bError:=fbReadVelocityToCam.bError OR fbReadVelocityFromCam.bError;
IF fbReadVelocityToCam.bError THEN
  nErrorId:=fbReadVelocityToCam.nErrorId;
ELSIF fbReadVelocityFromCam.bError THEN
  nErrorId:=fbReadVelocityFromCam.nErrorId;
END_IF

END_FUNCTION_BLOCK

// tc_mca_std_lib/POUs/ChangeConfig/FB_ReadFloatParameter
FUNCTION_BLOCK FB_ReadFloatParameter
VAR_INPUT
	bExecute: BOOL;
	///16#4000=Axisdata, 16#5000=Encoderdata, 16#6000=Controldata, 16#7000=Drivedata
	nDeviceGroup: UDINT;
	nIndexOffset: UDINT;
END_VAR
VAR_OUTPUT
	nData: LREAL;
	bBusy: BOOL;
	bDone: BOOL;
	bError: BOOL;
	nErrorId: UDINT;
END_VAR
VAR_IN_OUT
	Axis: AXIS_REF;
END_VAR
VAR
	nState: UINT;
	fbADSREAD: ADSREAD;
END_VAR

(*Sequence to read parameter in Nc*)
CASE nState OF
0:  (*Start sequence. Wait until bExecute is TRUE*)
	IF bExecute THEN
		bBusy:=TRUE;
		bError:=FALSE;
		nErrorId:=0;
		nState:=10;
	END_IF

10: (*Read parameter in Nc*)
	fbADSREAD(
		PORT:=500,
		IDXGRP:=nDeviceGroup+Axis.NcToPlc.AxisId,
		IDXOFFS:=nIndexOffset,
		LEN:=SIZEOF(nData),
		DESTADDR:=ADR(nData),
		READ:=TRUE);

	(*Wait until it's done or if an error occurs*)
	IF NOT fbADSREAD.ERR THEN
		IF NOT fbADSREAD.BUSY THEN
			fbADSREAD(READ:=FALSE);
			nState:=20;
		END_IF
	ELSE
		nErrorId:=fbADSREAD.ERRID;
		nState:=999;
	END_IF

20: (*Sequense is done. Waits until bExecute is FALSE*)
	bBusy:=FALSE;
	bDone:=TRUE;
	IF NOT bExecute THEN
		bDone:=FALSE;
		nState:=0;
	END_IF

999: (*Error in sequence*)
	bError:=TRUE;
	bBusy:=FALSE;
	bDone:=FALSE;
	fbADSREAD(READ:=FALSE);
	IF NOT bExecute THEN
		nState:=0;
	END_IF

END_CASE

END_FUNCTION_BLOCK

// tc_mca_std_lib/POUs/Motion/Homing/FB_HomeFinish
FUNCTION_BLOCK FB_HomeFinish
VAR_INPUT
	En: BOOL;
	bReset: BOOL;
    bExecute: BOOL;	
    nCmdData: UINT;
	bSofLimEnableLow: BOOL:=TRUE;
	bSofLimEnableHigh: BOOL:=TRUE;			
END_VAR
VAR_IN_OUT
	Axis: AXIS_REF;
END_VAR
VAR_OUTPUT
	EnO: BOOL;	
	bBusy: BOOL;
	bDone: BOOL;
	bError: BOOL;
	nErrorId: UDINT;
END_VAR
VAR		
	fbHomewriteSoftLimEnable:FB_HomeWriteSoftLimEnable;	
	fbExecuteRiseEdge: R_TRIG;	
	bExecuteWriteNC:BOOL:=FALSE;
	nState:INT:=0;
END_VAR

En:=EnO;
IF bReset THEN
	bError:=FALSE;
	nErrorId:=0;
END_IF 

IF NOT bExecute THEN
  bExecuteWriteNC:=FALSE;
  fbHomewriteSoftLimEnable.bSofLimEnableLow:=bSofLimEnableLow;
  fbHomewriteSoftLimEnable.bSofLimEnableHigh:=bSofLimEnableHigh;   
  nState:=0;
END_IF

fbExecuteRiseEdge(CLK:=bExecute);
IF fbExecuteRiseEdge.Q THEN
  bExecuteWriteNC:=TRUE;  
  fbHomewriteSoftLimEnable.bSofLimEnableLow:=bSofLimEnableLow;
  fbHomewriteSoftLimEnable.bSofLimEnableHigh:=bSofLimEnableHigh;
END_IF

// Write to NC (disable soft limits)
fbHomewriteSoftLimEnable(
	En:=En,
	bExecute:=bExecuteWriteNC AND bExecute,
	Axis:=Axis,
	bReset:=bReset,	
);

bBusy:=fbHomewriteSoftLimEnable.bBusy;
bDone:=fbHomewriteSoftLimEnable.bDone;

bError:=fbHomewriteSoftLimEnable.bError;
IF fbHomewriteSoftLimEnable.bError THEN
  nErrorId:=fbHomewriteSoftLimEnable.nErrorId;
END_IF

END_FUNCTION_BLOCK

// POUs/Motion/FB_MotionHoming
FUNCTION_BLOCK FB_MotionHoming
VAR_IN_OUT
    stMotionStage: DUT_MotionStage;
END_VAR
VAR_INPUT
    bExecute: BOOL;
END_VAR
VAR_OUTPUT
    bBusy: BOOL;
    bDone: BOOL;
    bError: BOOL;
    nErrorID: UDINT;
END_VAR
VAR
    fbSetPos: MC_SetPosition;
    fbJog: MC_Jog;
    rtExec: R_TRIG;
    ftExec: F_TRIG;
    nHomeStateMachine: INT := IDLE;
    nStateAfterStop: INT;
    nMoves: INT;
    bFirstDirection: BOOL;
    bAtHome: BOOL;
    bMove: BOOL;
    nErrCount: INT;
    bInterrupted: BOOL;
END_VAR
VAR CONSTANT
    IDLE: INT := 0;
    NEXT_MOVE: INT := 1;
    CHECK_FWD: INT := 2;
    CHECK_BWD: INT := 3;
    FINAL_MOVE: INT := 4;
    FINAL_SETPOS: INT := 5;
    ERROR: INT := 6;
    WAIT_STOP: INT := 7;

    (*
        This is a simpler way of disabling the soft limits that ends up being really obvious if something has gone wrong.
        If you turn the limits off/on, not only do you need to keep track of if you had soft limits set,
        but you need to always restore this properly or risk some issue.
        Instead, I set position to a ridiculous value that can always move forward or backward.
        If this gets stuck for any reason it's very clear that something has gone wrong,
        rather than a silent failure of the soft limit marks.
    *)
    FWD_START: LREAL := -99999999;
    BWD_START: LREAL :=  99999999;
END_VAR


fbSetPos.Options.ClearPositionLag := TRUE;
rtExec(CLK:=bExecute);
ftExec(CLK:=bExecute);

bError R= NOT bExecute;
IF NOT bError THEN
    nErrorID := 0;
END_IF

CASE stMotionStage.nHomingMode OF
    ENUM_EpicsHomeCmd.LOW_LIMIT:
        bFirstDirection := FALSE;
        bAtHome := NOT stMotionStage.bLimitBackwardEnable;
        bMove := TRUE;
    ENUM_EpicsHomeCmd.HIGH_LIMIT:
        bFirstDirection := TRUE;
        bAtHome := NOT stMotionStage.bLimitForwardEnable;
        bMove := TRUE;
    ENUM_EpicsHomeCmd.HOME_VIA_LOW:
        bFirstDirection := FALSE;
        bAtHome := stMotionStage.bHome;
        bMove := TRUE;
    ENUM_EpicsHomeCmd.HOME_VIA_HIGH:
        bFirstDirection := TRUE;
        bAtHome := stMotionStage.bHome;
        bMove := TRUE;
    ENUM_EpicsHomeCmd.ABSOLUTE_SET:
        fbSetPos(
            Axis:=stMotionStage.Axis,
            Execute:=bExecute,
            Position:=stMotionStage.fHomePosition);
        bBusy := rtExec.Q;
        bDone := NOT rtExec.Q;
        bMove := FALSE;
    ENUM_EpicsHomeCmd.NONE:
        bMove := FALSE;
        bBusy := rtExec.Q;
        bDone := NOT rtExec.Q;
    ELSE
        bMove := FALSE;
END_CASE

IF bMove THEN
    IF bBusy AND ftExec.Q THEN
        nHomeStateMachine := ERROR;
        bInterrupted := TRUE;
    END_IF
    CASE nHomeStateMachine OF
        // Wait for a rising edge
        IDLE:
            bBusy := FALSE;
            nErrCount := 0;
            fbSetPos(
                Axis:=stMotionStage.Axis,
                Execute:=FALSE);
            fbJog(
                Axis:=stMotionStage.Axis,
                JogForward:=FALSE,
                JogBackwards:=FALSE);
            IF rtExec.Q THEN
                nHomeStateMachine := NEXT_MOVE;
                nMoves := 0;
                bDone := FALSE;
                bBusy := TRUE;
                bError := FALSE;
                nErrorID := 0;
                bInterrupted := FALSE;
            END_IF
        // Figure out whether to move forward, move backward, or give up
        NEXT_MOVE:
            fbSetPos(
                Axis:=stMotionStage.Axis,
                Execute:=FALSE);
            fbJog(
                Axis:=stMotionStage.Axis,
                JogForward:=FALSE,
                JogBackwards:=FALSE);
            CASE nMoves OF
                0:
                    IF bFirstDirection THEN
                        nStateAfterStop := CHECK_FWD;
                    ELSE
                        nStateAfterStop := CHECK_BWD;
                    END_IF
                1:
                    IF NOT bFirstDirection THEN
                        nStateAfterStop := CHECK_FWD;
                    ELSE
                        nStateAfterStop := CHECK_BWD;
                    END_IF
                ELSE
                    nStateAfterStop := ERROR;
            END_CASE
            nMoves := nMoves + 1;
            IF bAtHome THEN
                nStateAfterStop := FINAL_MOVE;
            END_IF
            nHomeStateMachine := WAIT_STOP;
        // Move forward until we find the home signal or reach end of travel
        CHECK_FWD:
            fbSetPos(
                Axis:=stMotionStage.Axis,
                Execute:=TRUE,
                Position:=FWD_START);
            fbJog(
                Axis:=stMotionStage.Axis,
                JogForward:=stMotionStage.bLimitForwardEnable AND NOT bATHome,
                JogBackwards:=FALSE,
                Mode:=E_JogMode.MC_JOGMODE_CONTINOUS,
                Velocity:=stMotionStage.stAxisParameters.fRefVeloSearch);
            IF NOT fbJog.JogForward THEN
                nHomeStateMachine := NEXT_MOVE;
            ELSIF fbJog.Error THEN
                fbJog(
                    Axis:=stMotionStage.Axis,
                    JogForward:=FALSE,
                    JogBackwards:=FALSE);
                nErrCount := nErrCount + 1;
                IF nErrCount >= 3 THEN
                    nHomeStateMachine := ERROR;
                END_IF
            END_IF
        // Move backward until we find the home signal or reach end of travel
        CHECK_BWD:
            fbSetPos(
                Axis:=stMotionStage.Axis,
                Execute:=TRUE,
                Position:=BWD_START);
            fbJog(
                Axis:=stMotionStage.Axis,
                JogForward:=FALSE,
                JogBackwards:=stMotionStage.bLimitBackwardEnable AND NOT bATHome,
                Mode:=E_JogMode.MC_JOGMODE_CONTINOUS,
                Velocity:=stMotionStage.stAxisParameters.fRefVeloSearch);
            IF NOT fbJog.JogBackwards THEN
                nHomeStateMachine := NEXT_MOVE;
            ELSIF fbJog.Error THEN
                fbJog(
                    Axis:=stMotionStage.Axis,
                    JogForward:=FALSE,
                    JogBackwards:=FALSE);
                nErrCount := nErrCount + 1;
                IF nErrCount >= 3 THEN
                    nHomeStateMachine := ERROR;
                END_IF
            END_IF
        // Set position to get within soft lims, move slowly off signal
        FINAL_MOVE:
            fbSetPos(
                Axis:=stMotionStage.Axis,
                Execute:=TRUE,
                Position:=stMotionStage.fHomePosition);
            IF bAtHome THEN
                fbJog(
                    Axis:=stMotionStage.Axis,
                    JogForward:=NOT bFirstDirection,
                    JogBackwards:=bFirstDirection,
                    Mode:=E_JogMode.MC_JOGMODE_CONTINOUS,
                    Velocity:=stMotionStage.stAxisParameters.fRefVeloSync);
            ELSIF fbJog.Error THEN
                fbJog(
                    Axis:=stMotionStage.Axis,
                    JogForward:=FALSE,
                    JogBackwards:=FALSE);
                nErrCount := nErrCount + 1;
                IF nErrCount >= 3 THEN
                    nHomeStateMachine := ERROR;
                END_IF
            ELSE
                fbJog(
                    Axis:=stMotionStage.Axis,
                    JogForward:=FALSE,
                    JogBackwards:=FALSE);
                fbSetPos(
                    Axis:=stMotionStage.Axis,
                    Execute:=FALSE);
                nHomeStateMachine := WAIT_STOP;
                nStateAfterStop := FINAL_SETPOS;
            END_IF
        FINAL_SETPOS:
            fbSetPos(
                Axis:=stMotionStage.Axis,
                Execute:=TRUE,
                Position:=stMotionStage.fHomePosition);
            nHomeStateMachine := IDLE;
            bBusy := FALSE;
            bDone := TRUE;
        ERROR:
            bError := TRUE;
            nErrorID := fbJog.ErrorID;
            nHomeStateMachine := FINAL_SETPOS;
            fbSetPos(
                Axis:=stMotionStage.Axis,
                Execute:=FALSE);
            IF bInterrupted THEN
                stMotionStage.sCustomErrorMessage := 'Homing interrupted';
            ELSE
                stMotionStage.sCustomErrorMessage := 'Homing failure';
            END_IF
        WAIT_STOP:
            IF stMotionStage.Axis.Status.NotMoving THEN
                nHomeStateMachine := nStateAfterStop;
            END_IF
    END_CASE
END_IF

END_FUNCTION_BLOCK

// POUs/Motion/FB_EncSaveRestore
FUNCTION_BLOCK FB_EncSaveRestore
VAR_IN_OUT
    stMotionStage: DUT_MotionStage;
END_VAR
VAR_INPUT
    bEnable: BOOL;
END_VAR
VAR_OUTPUT
END_VAR
VAR
    fbSetPos: MC_SetPosition;
    timer: TON;
    bInit: BOOL;
    bLoad: BOOL;
    nLatchError: UDINT;
    bEncError: BOOL;
    tRetryDelay: TIME := T#1s;
    nMaxRetries: UINT := 10;
    nCurrTries: UINT := 0;
    bWaitRetry: BOOL;
    tonRetry: TON;
END_VAR
VAR PERSISTENT
    bSaved: BOOL;
    fPosition: LREAL;
END_VAR

IF bEnable THEN
    // Trigger a load if anything was saved at all
    IF NOT bInit THEN
        bInit := TRUE;
        bLoad S= bSaved;
        fbSetPos.Options.ClearPositionLag := TRUE;
    END_IF

    // Set our position if bLoad is true
    fbSetPos(
        Axis:=stMotionStage.Axis,
        Execute:=bLoad,
        Position:=fPosition);

    // Only load once, at startup
    bLoad R= fbSetPos.Done OR fbSetPos.Error;

    IF fbSetPos.Error THEN
        // Keep the error latched, it can disappear if Execute is set to FALSE
        nLatchError := fbSetPos.ErrorID;
        nCurrTries := nCurrTries + 1;
        IF nCurrTries >= nMaxRetries THEN
            // Alert the user that something has gone wrong
            stMotionStage.bError := TRUE;
            stMotionStage.nErrorId := nLatchError;
            stMotionStage.sCustomErrorMessage := 'Error loading previously saved position.';
        ELSE
            // Reset the FB for the next retry
            fbSetPos(
                Axis:=stMotionStage.Axis,
                Execute:=FALSE,
                Position:=fPosition);
            // Try again
            bWaitRetry := TRUE;
        END_IF
    END_IF

    tonRetry(
        IN := bWaitRetry,
        PT := tRetryDelay);

    bLoad S= tonRetry.Q;
    bWaitRetry R= tonRetry.Q;

    // Check DUT_MotionStage for an encoder error (range 0x44nn)
    bEncError := stMotionStage.bError AND stMotionStage.nErrorId >= 16#4400 AND stMotionStage.nErrorId <= 16#44FF;

    // Do not save if we're currently loading or if there is an encoder error
    IF NOT bLoad AND NOT bEncError AND NOT bWaitRetry THEN
        fPosition := stMotionStage.stAxisStatus.fActPosition;
        // This persistent variable lets us check if anything was saved
        // It will be TRUE at startup if we have saved values
        bSaved := TRUE;
    END_IF
END_IF

END_FUNCTION_BLOCK

// POUs/Motion/FB_LogMotionError
FUNCTION_BLOCK FB_LogMotionError
(*
    If the motion struct has an error, log it.

    The log condition is:
    - When bError goes TRUE (catch transition from no error to error)
    - When the error message changes while bError is TRUE (catch transition from error a to error b)

    Includes the motor name and the NC error id in the json blob
*)
VAR_IN_OUT
    stMotionStage: DUT_MotionStage;
END_VAR
VAR_INPUT
    bEnable: BOOL;
END_VAR
VAR
    fbLogMessage: FB_LogMessage;
    rtNewError: R_TRIG;
    bChangedError: BOOL;
    sPrevErr: STRING;
    fbJson: FB_JsonSaxWriter;
END_VAR


rtNewError(CLK:=stMotionStage.bError);
bChangedError := stMotionStage.sErrorMessage <> '' AND stMotionStage.sErrorMessage <> sPrevErr;
sPrevErr := stMotionStage.sErrorMessage;

IF bEnable AND (rtNewError.Q OR bChangedError) THEN
    fbJson.StartObject();
    fbJson.AddKey('schema');
    fbJson.AddString('DUT_MotionStage.bError');
    fbJson.AddKey('dut_name');
    fbJson.AddString(stMotionStage.sName);
    fbJson.AddKey('axis_name');
    fbJson.AddString(stMotionStage.stAxisParameters.sAxisName);
    fbJson.AddKey('axis_id');
    fbJson.AddUdint(stMotionStage.stAxisParameters.AxisId);
    fbJson.AddKey('err_id');
    fbJson.AddUdint(stMotionStage.nErrorId);
    fbJson.AddKey('position');
    fbJson.AddLreal(stMotionStage.stAxisStatus.fActPosition);
    fbJson.AddKey('position_lag');
    fbJson.AddLreal(stMotionStage.stAxisStatus.fActDiff);
    fbJson.EndObject();
    fbLogMessage.sJson := fbJson.GetDocument();
    fbLogMessage(
        sMsg := stMotionStage.sErrorMessage,
        eSevr := TcEventSeverity.Error,
        eSubsystem := E_Subsystem.MOTION,
    );
    fbJson.ResetDocument();
END_IF

END_FUNCTION_BLOCK

// POUs/Motion/Utils/FB_SetEnables
FUNCTION_BLOCK FB_SetEnables
// Update the all enable booleans based on the booleans that make them up
VAR_IN_OUT
    stMotionStage: DUT_MotionStage;
END_VAR

stMotionStage.bAllForwardEnable := stMotionStage.bLimitForwardEnable AND (stMotionStage.bGantryForwardEnable OR NOT stMotionStage.bGantryAxis) AND stMotionStage.stEPSForwardEnable.bEPS_OK;
stMotionStage.bAllBackwardEnable := stMotionStage.bLimitBackwardEnable AND (stMotionStage.bGantryBackwardEnable OR NOT stMotionStage.bGantryAxis) AND stMotionStage.stEPSBackwardEnable.bEPS_OK;

stMotionStage.bAllEnable := stMotionStage.bEnable AND stMotionStage.bHardwareEnable AND stMotionStage.stEPSPowerEnable.bEPS_OK;
stMotionStage.bAllEnable R= NOT stMotionStage.bUserEnable;

END_FUNCTION_BLOCK

// POUs/Motion/FB_EncoderValue
FUNCTION_BLOCK FB_EncoderValue
(*
    Process the encoder value for DUT_MotionStage

    A few different problems this is trying to solve:
        1. Different encoders show as different types in the IO,
           but we want a consistent type for checks and for PVs
        2. Some inverted encoders display as very high numbers
           as they count down from max int instead of up from 0
        3. Some encoders have raw signed values, others unsigned.

    To this end, we figure out which encoder is linked and process
    the value appropriately.
*)
VAR_IN_OUT
    stMotionStage: DUT_MotionStage;
END_VAR

IF stMotionStage.nRawEncoderULINT <> 0 THEN
    IF stMotionStage.nRawEncoderULINT < 4294967296 THEN
        stMotionStage.nEncoderCount := ULINT_TO_UDINT(stMotionStage.nRawEncoderULINT);
    ELSE
        stMotionStage.nEncoderCount := ULINT_TO_UDINT(18446744073709551615 - stMotionStage.nRawEncoderULINT);
    END_IF
ELSIF stMotionStage.nRawEncoderUINT <> 0 THEN
    stMotionStage.nEncoderCount := UINT_TO_UDINT(stMotionStage.nRawEncoderUINT);
ELSIF stMotionStage.nRawEncoderINT <> 0 THEN
    stMotionStage.nEncoderCount := INT_TO_UDINT(stMotionStage.nRawEncoderINT);
ELSE
    stMotionStage.nEncoderCount := 0;
END_IF

END_FUNCTION_BLOCK

// POUs/Motion/FB_MotionStageNCParams
FUNCTION_BLOCK FB_MotionStageNCParams
(*
    Read and refresh axis parameters struct on DUT_MotionStage
*)
VAR_IN_OUT
    stMotionStage: DUT_MotionStage;
END_VAR
VAR_INPUT
    bEnable: BOOL;
    tRefreshDelay: TIME;
END_VAR
VAR_OUTPUT
    bError: BOOL;
END_VAR
VAR
    mcReadParams: MC_ReadParameterSet;
    timer: TON;
    bExecute: BOOL := TRUE;
    nLatchErrId: UDINT;
END_VAR

timer(
    IN:=bEnable AND NOT bExecute,
    PT:=tRefreshDelay);
bExecute S= timer.Q;
mcReadParams(
    Parameter:=stMotionStage.stAxisParameters,
    Axis:=stMotionStage.Axis,
    Execute:=bEnable AND bExecute,
    Error=>bError);
IF mcReadParams.ErrorID <> 0 THEN
    nLatchErrId := 0;
END_IF
bExecute R= mcReadParams.Done OR mcReadParams.Error;
stMotionStage.bAxisParamsInit S= mcReadParams.Done;

END_FUNCTION_BLOCK

// POUs/Motion/States/Internals/FB_PositionStateInternal
FUNCTION_BLOCK FB_PositionStateInternal
(*
    Routines that must be called on all DUT_PositionState
*)
VAR_IN_OUT
    stMotionStage: DUT_MotionStage;
    stPositionState: DUT_PositionState;
END_VAR
VAR_OUTPUT
END_VAR
VAR
    fbEncConverter: FB_RawCountConverter;
    fbLock: FB_PositionStateLock;
END_VAR

// Mark that we've been here
stPositionState.bUpdated := TRUE;

// Update pos state's count or egu position as appropriate
IF stMotionStage.bAxisParamsInit THEN
    fbEncConverter(
        stParameters:=stMotionStage.stAxisParameters,
        nCountCheck:=stPositionState.nEncoderCount,
        fPosCheck:=stPositionState.fPosition);
    IF stPositionState.bUseRawCounts THEN
        stPositionState.fPosition := fbEncConverter.fPosGet;
    ELSE
        stPositionState.nEncoderCount := fbEncConverter.nCountGet;
    END_IF
END_IF

// Handle state parameter locking
fbLock(
    stPositionState:=stPositionState,
    bEnable:=stMotionStage.bAxisParamsInit);

END_FUNCTION_BLOCK

// POUs/Motion/States/Helpers/FB_RawCountConverter
FUNCTION_BLOCK FB_RawCountConverter
(*
    Utility function block for converting raw counts to EGU and back
*)
VAR_INPUT
    // Parameters to check against
    stParameters: ST_AxisParameterSet;
    // Optional count to convert to a real position
    nCountCheck: UDINT;
    // Optional position to convert to encoder counts
    fPosCheck: LREAL;
END_VAR
VAR_OUTPUT
    // If converting position, the number of counts
    nCountGet: UDINT;
    // If converting counts, the position
    fPosGet: LREAL;
    // True during a parameter get/calc
    bBusy: BOOL;
    // True after a successful get/calc
    bDone: BOOL;
    // True if the calculation errored
    bError: BOOL;
END_VAR

IF stParameters.fEncScaleFactorInternal <> 0 THEN
    nCountGet := LREAL_TO_UDINT((fPosCheck - stParameters.fEncOffset) / stParameters.fEncScaleFactorInternal);
    fPosGet := nCountCheck * stParameters.fEncScaleFactorInternal + stParameters.fEncOffset;
END_IF

END_FUNCTION_BLOCK

// POUs/Motion/States/Internals/FB_PositionStateLock
FUNCTION_BLOCK FB_PositionStateLock
(*
    Implements immutability for a locked DUT_PositionState
    Once this is called the first time, the parameters at the time of the call will be restored on all subsequent calls.
*)
VAR_IN_OUT
    stPositionState: DUT_PositionState;
END_VAR
VAR_INPUT
    bEnable: BOOL;
END_VAR
VAR
    stCachedPositionState: DUT_PositionState;
    bInit: BOOL := FALSE;
END_VAR

IF bEnable THEN
    // Force values to be cached if we've cached something
    IF bInit AND stPositionState.bLocked THEN
        stPositionState.sName := stCachedPositionState.sName;
        stPositionState.fPosition := stCachedPositionState.fPosition;
        stPositionState.fDelta := stCachedPositionState.fDelta;
        stPositionState.fVelocity := stCachedPositionState.fVelocity;
        stPositionState.fAccel := stCachedPositionState.fAccel;
        stPositionState.fDecel := stCachedPositionState.fDecel;
    // If we haven't cached and we should, make the cache. Note that we skip bLocked, bValid, and bMoveOk
    ELSIF NOT bInit AND stPositionState.bLocked THEN
        stCachedPositionState.sName := stPositionState.sName;
        stCachedPositionState.fPosition := stPositionState.fPosition;
        stCachedPositionState.fDelta := stPositionState.fDelta;
        stCachedPositionState.fVelocity := stPositionState.fVelocity;
        stCachedPositionState.fAccel := stPositionState.fAccel;
        stCachedPositionState.fDecel := stPositionState.fDecel;
        bInit := TRUE;
    // Do nothing, or unlock the state if bLocked goes FALSE
    ELSIF NOT stPositionState.bLocked THEN
        bInit := FALSE;
    END_IF
END_IF

END_FUNCTION_BLOCK

// POUs/Deprecated/FB_StatePTPMove
FUNCTION_BLOCK FB_StatePTPMove
// Do not use, this is deprecated
VAR_INPUT
    {attribute 'pytmc' := '
        pv:
    '}
    stPositionState: DUT_PositionState;

    {attribute 'pytmc' := '
        pv: GO
        io: io
        field: ZNAM False
        field: ONAM True
    '}
    bExecute: BOOL;

    bMoveOk: BOOL;
END_VAR
VAR_IN_OUT
    stMotionStage: DUT_MotionStage;
END_VAR
VAR_OUTPUT
    {attribute 'pytmc' := '
        pv: AT_STATE
        io: input
        field: ZNAM False
        field: ONAM True
    '}
    bAtState: BOOL;

    {attribute 'pytmc' := '
        pv: DMOV
        io: input
        field: ZNAM False
        field: ONAM True
    '}
    bDone: BOOL;

    {attribute 'pytmc' := '
        pv: BUSY
        io: input
        field: ZNAM False
        field: ONAM True
    '}
    bBusy: BOOL;

    {attribute 'pytmc' := '
        pv: ERR
        io: input
        field: ZNAM False
        field: ONAM True
    '}
    bError: BOOL;

    {attribute 'pytmc' := '
        pv: ERRMSG
        io: input
    '}
    sError: STRING;
END_VAR
VAR
    bExecTrig: R_TRIG;
    bExecEnd: F_TRIG;
    fActPosition: LREAL;
    fLowPos: LREAL;
    fHighPos: LREAL;
END_VAR

bExecTrig(CLK:=bExecute);
IF bExecTrig.Q AND bMoveOk THEN
    IF NOT stMotionStage.bBusy AND NOT stMotionStage.bError THEN
        stMotionStage.bExecute := TRUE;
        stMotionStage.nCommand := ENUM_EpicsMotorCmd.MOVE_ABSOLUTE;
        stMotionStage.fPosition := stPositionState.fPosition;
        stMotionStage.fVelocity := stPositionState.fVelocity;
        stMotionStage.fAcceleration := stPositionState.fAccel;
        stMotionStage.fDeceleration := stPositionState.fDecel;
        bDone := FALSE;
        bBusy := TRUE;
    END_IF
END_IF
bError := stMotionStage.bError;
sError := stMotionStage.sErrorMessage;

fActPosition := stMotionStage.stAxisStatus.fActPosition;
fLowPos := stPositionState.fPosition - stPositionState.fDelta;
fHighPos := stPositionState.fPosition + stPositionState.fDelta;
IF (fLowPos < fActPosition) AND (fHighPos > fActPosition) THEN
    bAtState := TRUE;
    IF NOT stMotionStage.bBusy THEN
        bDone := TRUE;
        bBusy := FALSE;
        bExecute := FALSE;
    END_IF
ELSE
    bAtState := FALSE;
END_IF

bExecEnd(CLK:=bExecute);
IF bExecEnd.Q AND bBusy THEN
    stMotionStage.bExecute := FALSE;
END_IF

IF NOT stMotionStage.bExecute OR NOT bExecute THEN
    bDone := TRUE;
    bBusy := FALSE;
    bExecute := FALSE;
END_IF

END_FUNCTION_BLOCK

// POUs/ImplicitChecks/CheckBounds
// Implicitly generated code : DO NOT EDIT
FUNCTION CheckBounds : DINT
VAR_INPUT
    index, lower, upper: DINT;
END_VAR

// Implicitly generated code : Only an Implementation suggestion
{noflow}
IF  index < lower THEN
    CheckBounds := lower;
ELSIF  index > upper THEN
    CheckBounds := upper;
ELSE
    CheckBounds := index;
END_IF
{flow}

END_FUNCTION

// POUs/ImplicitChecks/CheckDivDInt
// Implicitly generated code : DO NOT EDIT
FUNCTION CheckDivDInt : DINT
VAR_INPUT
    divisor:DINT;
END_VAR

// Implicitly generated code : Only an Implementation suggestion
{noflow}
IF divisor = 0 THEN
    CheckDivDInt:=1;
ELSE
    CheckDivDInt:=divisor;
END_IF;
{flow}

END_FUNCTION

// POUs/ImplicitChecks/CheckDivLInt
// Implicitly generated code : DO NOT EDIT
FUNCTION CheckDivLInt : LINT
VAR_INPUT
    divisor:LINT;
END_VAR

// Implicitly generated code : Only an Implementation suggestion
{noflow}
IF divisor = 0 THEN
    CheckDivLInt:=1;
ELSE
    CheckDivLInt:=divisor;
END_IF;
{flow}

END_FUNCTION

// POUs/ImplicitChecks/CheckDivLReal
// Implicitly generated code : DO NOT EDIT
FUNCTION CheckDivLReal : LREAL
VAR_INPUT
    divisor:LREAL;
END_VAR

// Implicitly generated code : Only an Implementation suggestion
{noflow}
IF divisor = 0 THEN
    CheckDivLReal:=1;
ELSE
    CheckDivLReal:=divisor;
END_IF;
{flow}

END_FUNCTION

// POUs/ImplicitChecks/CheckDivReal
// Implicitly generated code : DO NOT EDIT
FUNCTION CheckDivReal : REAL
VAR_INPUT
    divisor:REAL;
END_VAR

// Implicitly generated code : Only an Implementation suggestion
{noflow}
IF divisor = 0 THEN
    CheckDivReal:=1;
ELSE
    CheckDivReal:=divisor;
END_IF;
{flow}

END_FUNCTION

// POUs/Motion/Gantry/FB_GantryAutoCoupling
FUNCTION_BLOCK FB_GantryAutoCoupling
VAR_INPUT
    nGantryTol : LINT;
END_VAR
VAR_OUTPUT
    bGantryAlreadyCoupled : BOOL;
END_VAR
VAR_IN_OUT
    Master : DUT_MotionStage;
    MasterEnc : ST_RenishawAbsEnc;
    Slave : DUT_MotionStage;
    SlaveEnc : ST_RenishawAbsEnc;
    bExecuteCouple : BOOL;
    bExecuteDecouple : BOOL;
END_VAR
VAR
    gantry_diff_limit : FB_GantryDiffVirtualLimitSwitch;
    couple : MC_GEARIN;
    decouple : MC_GEAROUT;
    bInitComplete : BOOL;
    fbSetEnables : FB_SetEnables;
END_VAR

// Designate Master and SLave Axes
Master.bGantryAxis := TRUE;
Slave.bGantryAxis := TRUE;

Master.nGantryTol := nGantryTol;
Slave.nGantryTol := Master.nGantryTol;

// Activate Gantry Virtual Limit Switch
gantry_diff_limit(Penc:=MasterEnc, SEnc:=SlaveEnc, GantDiffTol:=Master.nGantryTol,
                  PLimFwd=>Master.bGantryForwardEnable, PLimBwd=>Master.bGantryBackwardEnable,
                  SLimFwd=>Slave.bGantryForwardEnable, SLimBwd=>Slave.bGantryBackwardEnable);

// Coupling Status Bit
bGantryAlreadyCoupled := Master.Axis.NcToPlc.CoupleState=1 AND Slave.Axis.NcToPlc.CoupleState=3;

fbSetEnables(stMotionStage:=Master);
fbSetEnables(stMotionStage:=Slave);

IF bGantryAlreadyCoupled THEN
    Master.bGantryForwardEnable := Master.bGantryForwardEnable AND Slave.bAllForwardEnable;
    Slave.bGantryForwardEnable := Master.bAllForwardEnable AND Slave.bGantryForwardEnable;

    Master.bGantryBackwardEnable := Master.bGantryBackwardEnable AND Slave.bAllBackwardEnable;
    Slave.bGantryBackwardEnable := Master.bAllBackwardEnable AND Slave.bGantryBackwardEnable;
END_IF


// Coupling states
// Auto-coupling at init and auto-reset of coupling boolean
bExecuteCouple S= NOT bInitComplete;

bExecuteCouple R= couple.Busy OR bGantryAlreadyCoupled;
couple(Master:=Master.Axis, Slave:=Slave.Axis, Execute:=bExecuteCouple);

bInitComplete S= bGantryAlreadyCoupled;

// Decoupling with auto-reset of coupling boolean
bExecuteDecouple R= decouple.Busy OR NOT bGantryAlreadyCoupled;
decouple(Slave:=Slave.Axis, Execute:=bExecuteDecouple);

END_FUNCTION_BLOCK

// POUs/Motion/Gantry/FB_GantryDiffVirtualLimitSwitch
FUNCTION_BLOCK FB_GantryDiffVirtualLimitSwitch
VAR_INPUT
    PEnc: ST_RenishawAbsEnc; // Primary axis encoder (usually the upstream one)
    SEnc: ST_RenishawAbsEnc; // Secondary axis encoder (couples to the primary)

    GantDiffTol: LINT;        // Gantry differenace tolerance in encoder counts
END_VAR
VAR_OUTPUT
    PLimFwd: BOOL; // Primary axis forward direction enable
    PLimBwd: BOOL; // Primary axis reverse direction enable
    SLimFwd: BOOL; // Secondary axis forward direction enable
    SLimBwd: BOOL; // Secondary axis reverse direction enable
END_VAR
VAR
    GantryDiff: LINT;
END_VAR

(* Gantry Difference Virtual Limit Switch
A. Wallace 2017-2-15

Determines which direction is disabled due to it increasing the gantry difference.
Refer to the ESD for actual conventions.

A positive gantry error refers to a CCW clocked assembly:
eg. for X
X1 upstream, X2 downstream. Primary axis is always upstream.
Gantry difference > 0 when
X2>X1
Therefore
X2 positive direction disabled
X1 negative direction disabled

Call before FB_MotionStage fb calls for the gantry axes.
*)

GantryDiff := ( ULINT_TO_LINT(PEnc.Count) - ULINT_TO_LINT(PEnc.Ref) ) - ( ULINT_TO_LINT(SEnc.Count) - ULINT_TO_LINT(SEnc.Ref) );

IF ABS(GantryDiff) > GantDiffTol THEN
    IF GantryDiff < 0  THEN
        PLimBwd := FALSE;
        SLimFwd := FALSE;
    ELSE
        PLimBwd := TRUE;
        SLimFwd := TRUE;
    END_IF
    IF GantryDiff > 0 THEN
        PLimFwd := FALSE;
        SLimBwd := FALSE;
    ELSE
        PLimFwd := TRUE;
        SLimBwd := TRUE;
    END_IF
ELSE
    //If there is no fault, all directions are enabled
    PLimFwd := TRUE;
    PLimBwd := TRUE;
    SLimFwd := TRUE;
    SLimBwd := TRUE;
END_IF

END_FUNCTION_BLOCK

// POUs/Motion/PMPS/FB_EncErrorFFO
FUNCTION_BLOCK FB_EncErrorFFO
(*
    Example usage of FB_NCErrorFFO that only counts encoder errors as faults.
*)
VAR_IN_OUT
    // Motion stage to monitor
    stMotionStage: DUT_MotionStage;
    // FFO to trip
    fbFFHWO: FB_HardwareFFOutput;
END_VAR
VAR_INPUT
    // Reset the fault
    bReset: BOOL;
    // Auto reset the fault
    bAutoReset: BOOL;
END_VAR
VAR_OUTPUT
    // Quick way for nearby code to check if this block has tripped the FFO.
    bTripped: BOOL;
END_VAR
VAR
    fbNCErrorFFO: FB_NCErrorFFO := (
        nLowErrorId := 16#4400,
        nHighErrorId := 16#44FF,
        sDesc := 'Encoder error');
END_VAR

fbNCErrorFFO(
    stMotionStage := stMotionStage,
    fbFFHWO := fbFFHWO,
    bReset := bReset,
    bAutoReset := bAutoReset,
    bTripped => bTripped);

END_FUNCTION_BLOCK

// POUs/Motion/PMPS/FB_NCErrorFFO
FUNCTION_BLOCK FB_NCErrorFFO
(*
    Configure a DUT_MotionStage to trigger an FFO when we have an error.

    This can be configured to only apply to specific error ranges,
    though the default is the normal 16#4XXX NC error range. The error
    ranges are:
    16#40XX General Errors
    16#41XX Channel Errors
    16#42XX Group Errors
    16#43XX Axis Errors
    16#44XX Encoder Errors
    16#45XX Controller Errors
    16#46XX Drive Errors
    16#4AXX Table Errors
    16#4BXX NC PLC Errors
    16#4CXX Kinematic Transformation

    There is also a new extended NC error range, but it is sparsely populated.
    This range is 16#8XXX:
    16#8100 - 16#811F: Bode plot (diagnosis)
    16#8120 - 16#8FFF: Further errors

    To configure multiple ranges, simply use multiple instances of this
    function block.
*)
VAR_IN_OUT
    // Motion stage to monitor
    stMotionStage: DUT_MotionStage;
    // FFO to trip
    fbFFHWO: FB_HardwareFFOutput;
END_VAR
VAR_INPUT
    // Reset the fault
    bReset: BOOL;
    // Auto-reset the fault
    bAutoReset: BOOL;
    // The lowest error code that will trip the FFO
    nLowErrorId: UDINT := 16#4000;
    // The highest error code that will trip the FFO
    nHighErrorId: UDINT := 16#4FFF;
    // A description of the fault
    sDesc: STRING := 'Motor error';
END_VAR
VAR_OUTPUT
    // Quick way for nearby code to check if this block has tripped the FFO.
    bTripped: BOOL;
    // Error code sent to PMPS. Is always 16#20XX, where XX is the first two hex in the NC error.
    nErrorTypeCode: UINT;
END_VAR
VAR
    bInit: BOOL := TRUE;
    bNCError: BOOL;
    stBeamParams: ST_BeamParams;
    fbFF: FB_FastFault;
    rtTrip: R_TRIG;
END_VAR

IF bInit THEN
    fbFF.i_DevName := stMotionStage.sName;
    fbFF.i_Desc := sDesc;
    IF LEN(stMotionStage.sName) > 0 THEN
        bInit := FALSE;
    END_IF
ELSE
    bNCError := stMotionStage.bError AND stMotionStage.nErrorId >= nLowErrorId AND stMotionStage.nErrorId <= nHighErrorId;
    bTripped := bNCError AND PMPS_GVL.stCurrentBeamParameters.nRate > 0;
    rtTrip(CLK:=bTripped);
    IF rtTrip.Q THEN
        nErrorTypeCode := 16#2000 + UDINT_TO_UINT(SHR(stMotionStage.nErrorId, 8));
    END_IF
    fbFF(i_xOK := NOT bTripped,
         i_xReset := bReset,
         i_xAutoReset := bAutoReset,
         i_TypeCode:= nErrorTypeCode,
         io_fbFFHWO := fbFFHWO);
END_IF

END_FUNCTION_BLOCK

// POUs/Motion/PMPS/FB_PositionStatePMPS
FUNCTION_BLOCK FB_PositionStatePMPS EXTENDS FB_PositionStatePMPS_Base
(*
    Hooks up a position state to an arbiter and an FFO
        Use BeamParameterTransitionManager to manage transition requests between states
        Hook up to the inputs/outputs of the state function block
        Raises FFO if beam parameters are worse than required for current state
*)
VAR_IN_OUT
    fbArbiter: FB_Arbiter;
    fbFFHWO: FB_HardwareFFOutput;
END_VAR
VAR_INPUT
    bReadPmpsDb: BOOL;
    sPmpsDeviceName: STRING;
    sTransitionKey: STRING;
    stPmpsDoc: SJsonValue;
    stHighBeamThreshold: ST_BeamParams := PMPS_GVL.cstFullBeam;
    bBPOKAutoReset: BOOL := False;
END_VAR
VAR
    arrPMPS: ARRAY[0..GeneralConstants.MAX_STATES] OF ST_DbStateParams;
    nBPIndex: INT;
    nTransitionAssertionID: UDINT;
    nLastReqAssertionID: UDINT;
    fbReadPmpsDb: FB_JsonDocToSafeBP;
    ftDbBusy: F_TRIG;
    rtReadDBExec: R_TRIG;
    ftRead: F_TRIG;
    bptm: BeamParameterTransitionManager;
    ffBeamParamsOk: FB_FastFault;
    ffZeroRate: FB_FastFault;
    ffBPTMTimeoutAndMove: FB_FastFault;
    ffBPTMError: FB_FastFault;
    ffMaint: FB_FastFault;
    ffUnknown: FB_FastFault;
    bFFOxOk: BOOL;
    bAtSafeState: BOOL;
    nIter: INT;
END_VAR

Exec();

ACTION AssertHere:
fbArbiter.AddRequest(
    sDevName := stMotionStage.sName,
    nReqID := stStateReq.stPMPS.nRequestAssertionID,
    stReqBP := stStateReq.stPMPS.stBeamParams);
END_ACTION

ACTION ClearAsserts:
fbArbiter.RemoveRequest(nTransitionAssertionID);
FOR nIter := 1 TO GeneralConstants.MAX_STATES DO
    fbArbiter.RemoveRequest(arrStates[nIter].stPMPS.nRequestAssertionID);
END_FOR
END_ACTION

ACTION HandleBPTM:
(*
  Handle finishing the bptm late if timed out
  bptm needs a rising edge of bTransDone after authorizing transition
  If we fall into this block, bTransDone would otherwise be stuck at TRUE forever
  so the BPTM would never see a rising edge and therefore stay stuck
  We set to FALSE here to reset the BPTM, then gets set to TRUE again if really done.
*)
rtDoLateFinish(CLK:=bLateFinish AND bInternalAuth);
IF rtDoLateFinish.Q THEN
    bTransDone := FALSE;
    bLateFinish := FALSE;
END_IF

IF stStateReq.stPMPS.nRequestAssertionID <> nTransitionAssertionID THEN
    (*
        Edge case: the request is swapped out without a move
        Same as above: we need a rising edge of bTransDone, so cause a falling edge and the let the rising edge happen next cycle
        This will already be false when we request a positional move
    *)
    bTransDone R= stStateReq.stPMPS.nRequestAssertionID <> nLastReqAssertionID;
    // Just normal bptm call
    bptm(fbArbiter:=fbArbiter,
         i_sDeviceName:=stMotionStage.sName,
         i_TransitionAssertionID:=nTransitionAssertionID,
         i_stTransitionAssertion:=stTransitionBeam,
         i_nRequestedAssertionID:=stStateReq.stPMPS.nRequestAssertionID,
         i_stRequestedAssertion:=stStateReq.stPMPS.stBeamParams,
         i_xDoneMoving:=bTransDone,
         stCurrentBeamParameters:=PMPS_GVL.stCurrentBeamParameters,
         q_xTransitionAuthorized=>bInternalAuth,
         bDone=>bBPTMDone);
    nLastReqAssertionID := stStateReq.stPMPS.nRequestAssertionID;
END_IF
END_ACTION

ACTION HandleFFO:
// stBeamNeeded will point to Unknown/No beam if we are out of state bounds or in motion
// Otherwise we'll have the current state's beam parameters

// Check for bad conditions
bFFOxOk := F_SafeBPCompare(PMPS_GVL.stCurrentBeamParameters, stBeamNeeded);
// It is safe to reset automatically if our current state can take full beam.
// Otherwise we'll have to ask for a user acknowledgement to clear.
// This avoids rapidly cycling the FFOs on/off
// You can pass in a different stHighBeamThreshold as an input parameter to customize this behavior
bAtSafeState := F_SafeBPCompare(stHighBeamThreshold, stBeamNeeded);

// If the beam parameters are wrong, it is a fault! This encompasses all unknown arbiter-related errors.
ffBeamParamsOk.i_xOK := bFFOxOk;
ffBeamParamsOk.i_xReset S= bFFOxOk AND bAtSafeState;
ffBeamParamsOk.i_xReset R= NOT ffBeamParamsOk.i_xOK;
ffBeamParamsOk.i_xAutoReset := bBPOKAutoReset;

ffBeamParamsOk(
    i_DevName:=stMotionStage.sName,
    i_Desc:='Beam parameter mismatch',
    i_TypeCode:=16#1000,
    io_fbFFHWO:=fbFFHWO);

// Trip the beam for zero-rate states. This is a PMPS training wheel and should ultimately be removed.
// Note: I think this is already redundant
ffZeroRate(
    i_xOk := stBeamNeeded.nRate > 0,
    i_xAutoReset := TRUE,
    i_DevName := stMotionStage.sName,
    i_Desc := 'Device requesting zero rate',
    i_TypeCode := 16#1001,
    io_fbFFHWO := fbFFHWO);

// Trip the beam for BPTM timeouts if we want to move
// Only reset at safe beam OR at no bptm errors (some other FF should catch additional issues)
ffBPTMTimeoutAndMove.i_xOK := NOT (bArbiterTimeout AND bMoveOnArbiterTimeout);
ffBPTMTimeoutAndMove.i_xReset S= bAtSafeState OR (bptm.bDone AND NOT bptm.bError);
ffBPTMTimeoutAndMove.i_xReset R= NOT ffBPTMTimeoutAndMove.i_xOK;
ffBPTMTimeoutAndMove(
    i_DevName := stMotionStage.sName,
    i_Desc := 'BPTM Timeout',
    i_TypeCode := 16#1002,
    io_fbFFHWO := fbFFHWO);

// Trip the beam for BPTM Errors
ffBPTMError.i_xOK := NOT bptm.bError;
ffBPTMError.i_xReset S= bptm.bDone AND NOT bptm.bError;
ffBPTMError.i_xReset R= NOT ffBPTMError.i_xOK;
ffBPTMError(
    i_DevName := stMotionStage.sName,
    i_Desc := 'BPTM error, state transition failed',
    i_TypeCode := 16#1003,
    io_fbFFHWO := fbFFHWO);

// Trip the beam for maintenance mode
ffMaint(
    i_xOK := NOT bMaintMode,
    i_xAutoReset := TRUE,
    i_DevName := stMotionStage.sName,
    i_Desc := 'Device is in maintenance mode',
    i_TypeCode := 16#1004,
    io_fbFFHWO := fbFFHWO);

// Trip the beam for unknown state
ffUnknown(
    i_xOK := getState > 0 OR bInTransition,
    i_xAutoReset := TRUE,
    i_DevName := stMotionStage.sName,
    i_Desc := 'Unknown position between moves',
    i_TypeCode := 16#1005,
    io_fbFFHWO := fbFFHWO);
END_ACTION

ACTION HandlePmpsDb:

// Automatically read from the pmps db when it updates
// Assume update if no longer busy and no errors

ftDbBusy(CLK:=MOTION_GVL.fbPmpsFileReader.bBusy);
IF ftDbBusy.Q THEN
    bReadPmpsDb S= NOT MOTION_GVL.fbPmpsFileReader.bError;
END_IF

rtReadDBExec(CLK:=bReadPmpsDb);
IF rtReadDBExec.Q THEN
    arrPMPS[0].sPmpsState := sTransitionKey;
    FOR nBPIndex := 1 TO GeneralConstants.MAX_STATES BY 1 DO
        arrPMPS[nBPIndex] := arrStates[nBPIndex].stPMPS;
    END_FOR
END_IF

fbReadPmpsDb(
    bExecute:=bReadPmpsDb,
    jsonDoc:=stPmpsDoc,
    sDeviceName:=sPmpsDeviceName,
    io_fbFFHWO:=fbFFHWO,
    arrStates:=arrPMPS,
);
bReadPmpsDb R= NOT fbReadPmpsDb.bBusy;

ftRead(CLK:=fbReadPmpsDb.bBusy);

stTransitionState.sName := 'Transition';
IF ftRead.Q AND NOT fbReadPmpsDb.bError THEN
    stTransitionDb := arrPMPS[0];
    stTransitionBeam := arrPMPS[0].stBeamParams;
    nTransitionAssertionID := arrPMPS[0].nRequestAssertionID;
    stTransitionState.stPMPS := arrPMPS[0];
    FOR nBPIndex := 1 TO GeneralConstants.MAX_STATES BY 1 DO
        arrStates[nBPIndex].stPMPS := arrPMPS[nBPIndex];
    END_FOR
END_IF
END_ACTION

END_FUNCTION_BLOCK

// POUs/Motion/PMPS/FB_PositionStatePMPS_Base
FUNCTION_BLOCK FB_PositionStatePMPS_Base
(*
    FB_PositionStatePMPS without Arbiter, BPTM, FFO

    This allows me to test most of the code without an arbiter plc setup
*)
VAR_IN_OUT
    stMotionStage: DUT_MotionStage;
    arrStates: ARRAY[1..GeneralConstants.MAX_STATES] OF DUT_PositionState;
END_VAR
VAR_INPUT
    bArbiterEnabled: BOOL := TRUE;
    {attribute 'pytmc' := '
        pv: MAINT
        io: io
    '}
    bMaintMode: BOOL;
    bRequestTransition: BOOL;
    setState: INT;
    getState: INT;
    fStateBoundaryDeadband: LREAL := 0;
    tArbiterTimeout: TIME := T#1s;
    bMoveOnArbiterTimeout: BOOL := TRUE;
END_VAR
VAR_OUTPUT
    bTransitionAuthorized: BOOL;
    bForwardAuthorized: BOOL;
    bBackwardAuthorized: BOOL;
    bArbiterTimeout: BOOL;
END_VAR
VAR
    {attribute 'pytmc' := '
        pv: TRANS
        io: i
    '}
    stTransitionDb: ST_DbStateParams;
    stTransitionBeam: ST_BeamParams := PMPS_GVL.cst0RateBeam;
    stTransitionState: DUT_PositionState;
    bInit: BOOL := TRUE;
    bTransDone: BOOL;
    rtTransReq: R_TRIG;
    bBPTMDone: BOOL;
    rtBPTMDone: R_TRIG;
    ftMotorExec: F_TRIG;
    rtTransDone: R_TRIG;
    rtDoLateFinish: R_TRIG;
    tonDone: TON;
    stStateReq: DUT_PositionState;
    mcPower: MC_POWER;
    fUpperBound: LREAL;
    fLowerBound: LREAL;
    nGoalState: INT;
    stGoalState: DUT_PositionState;
    fActPos: LREAL;
    fReqPos: LREAL;
    bInTransition: BOOL;
    stBeamNeeded: ST_BeamParams;
    bFwdOk: BOOL;
    bBwdOk: BOOL;
    tonArbiter: TON;
    bLateFinish: BOOL;
    bInternalAuth: BOOL;
END_VAR

// This is meant to be subclassed. The parent class body is in the Exec action.

ACTION AssertHere:

END_ACTION

ACTION ClearAsserts:

END_ACTION

ACTION Exec:

// Load the pmps parameters as needed
HandlePmpsDb();

// Initialize or reinitialize to the current state value
rtBPTMDone(CLK:=bBPTMDone);
ftMotorExec(CLK:=stMotionStage.bExecute);
tonDone(
    IN:=bTransDone,
    PT:=T#100ms
    );
IF rtBPTMDone.Q OR ftMotorExec.Q OR tonDone.Q THEN
    bInit := TRUE;
END_IF
IF bInit OR nGoalState = 0 OR stMotionStage.bError THEN
    bInit R= stMotionStage.bAxisParamsInit;
    nGoalState := getState;
    stStateReq := GetStateStruct(getState);
    bInTransition := FALSE;
    rtTransReq(CLK:=FALSE);
    bTransitionAuthorized := FALSE;
    bArbiterTimeout := FALSE;
END_IF

// Request transition on rising edge
rtTransReq(CLK:=bRequestTransition);
IF rtTransReq.Q THEN
    nGoalState := setState;
    stStateReq := GetStateStruct(setState);
    bInTransition := TRUE;
    bTransDone := FALSE;
ELSE
    bTransDone := F_AtPositionState(stMotionStage:=stMotionStage, stPositionState:=stStateReq) AND NOT stMotionStage.bBusy;
END_IF

// Mark late finish if bTransDone -> true before the bptm is done
// This means that we finished the move so fast that the bptm needs to be unstuck via toggling bTransDone
rtTransDone(CLK:=bTransDone);
bLateFinish S= rtTransDone.Q AND NOT bBPTMDone;

IF bArbiterEnabled THEN
    // Handles getting the request to the arbiter and back
    HandleBPTM();
    // Handle arbiter timeouts
    IF tArbiterTimeout > T#0s THEN
        tonArbiter(
            IN:=bInTransition AND NOT bInternalAuth,
            PT:=tArbiterTimeout,
            Q=>bArbiterTimeout);
    ELSE
        bArbiterTimeout := FALSE;
    END_IF
    bTransitionAuthorized S= bInternalAuth OR (bArbiterTimeout AND bMoveOnArbiterTimeout);
ELSE
    // Clear all of our assertions if we decide to disable the arbiter
    ClearAsserts();
    // Do some dummy request handling
    bTransitionAuthorized := stMotionStage.bExecute;
    bArbiterTimeout := stMotionStage.bExecute;
END_IF

// Set up MPS virtual limit for moves at and between states
stGoalState := GetStateStruct(nGoalState);
fActPos := stMotionStage.stAxisStatus.fActPosition;
IF stMotionStage.bExecute THEN
    fReqPos := stMotionStage.fPosition;
ELSE
    fReqPos := fActPos;
END_IF

// Start with no move authority
bForwardAuthorized := FALSE;
bBackwardAuthorized := FALSE;

// Check if it would be OK to move without granting auth
bFwdOk := F_PosUnderUpperBound(MAX(fActPos, fReqPos) + ABS(fStateBoundaryDeadband), stGoalState);
bBwdOk := F_PosOverLowerBound(MIN(fActPos, fReqPos) - ABS(fStateBoundaryDeadband), stGoalState);

// Grant auth during moves based on goal state, current position, and goal position
IF stMotionStage.bExecute AND stGoalState.bValid THEN
    bForwardAuthorized := bFwdOk;
    bBackwardAuthorized := bBwdOk;
END_IF

IF bInTransition THEN
    // Deny auth during a transition request until transition is authorized
    bForwardAuthorized R= NOT bTransitionAuthorized;
    bBackwardAuthorized R= NOT bTransitionAuthorized;
    // Have the motor wait for permission to start move instead of immediately erroring
    stMotionStage.bSafetyReady := bTransitionAuthorized;
ELSE
    // If not transitioning, no need to wait for safety: immediately try to move and error if no auth
    stMotionStage.bSafetyReady := stMotionStage.bExecute;
    // Set an error message override in case this causes an error
    IF stMotionStage.bError AND bArbiterEnabled AND NOT bMaintMode THEN
        IF fReqPos > fActPos AND NOT bFwdOk THEN
            stMotionStage.sCustomErrorMessage := 'Unsafe tweak forward blocked by PMPS';
        ELSIF fReqPos < fActPos AND NOT bBwdOk THEN
            stMotionStage.sCustomErrorMessage := 'Unsafe tweak backward blocked by PMPS';
        END_IF
    END_IF
END_IF

IF bArbiterEnabled AND NOT bMaintMode THEN
// Only let us move if the transition is allowed, or if we are moving within a state's bounds
    mcPower(Axis:=stMotionStage.Axis,
            Enable:=stMotionStage.bAllEnable,
            Enable_Positive:=stMotionStage.bAllForwardEnable AND bForwardAuthorized,
            Enable_Negative:=stMotionStage.bAllBackwardEnable AND bBackwardAuthorized);
ELSE
    mcPower(Axis:=stMotionStage.Axis,
            Enable:=stMotionStage.bAllEnable,
            Enable_Positive:=stMotionStage.bAllForwardEnable,
            Enable_Negative:=stMotionStage.bAllBackwardEnable);
    stMotionStage.bSafetyReady := TRUE;
END_IF

// Raise fast faults as needed
stBeamNeeded := GetBeamFromState(getState);
HandleFFO();
END_ACTION

METHOD GetBeamFromState : ST_BeamParams;
VAR_INPUT
    nState: INT;
END_VAR
VAR
    stState: DUT_PositionState;
END_VAR
stState := GetStateStruct(nState);
GetBeamFromState := stState.stPMPS.stBeamParams;
END_METHOD

METHOD GetStateCode : INT
VAR_INPUT
    nState: INT;
END_VAR
IF nState < 0 OR nState > GeneralConstants.MAX_STATES THEN
    GetStateCode := -1;
ELSE
    GetStateCode := nState;
END_IF
END_METHOD

METHOD GetStateStruct : DUT_PositionState
VAR_INPUT
    nState: INT;
END_VAR
{warning disable C0371}
// Implicit VAR_IN_OUT reference inside a method needs special handling
IF NOT __ISVALIDREF(arrStates) THEN
    GetStateStruct := stTransitionState;
    RETURN;
END_IF
CASE GetStateCode(nState) OF
    -1: GetStateStruct := stTransitionState;
    0: GetStateStruct := stTransitionState;
    ELSE
        GetStateStruct := arrStates[nState];
END_CASE
{warning restore C0371}
END_METHOD

ACTION HandleBPTM:

END_ACTION

ACTION HandleFFO:

END_ACTION

ACTION HandlePmpsDb:

END_ACTION

END_FUNCTION_BLOCK

// POUs/Motion/PMPS/FB_PositionStatePMPS_Test
FUNCTION_BLOCK FB_PositionStatePMPS_Test EXTENDS FB_PositionStatePMPS_Base
(*
    Implement position state pmps with no FFO and auto-accept transition after 3s
    Use for offline testing of everything except the explicit interface
*)
VAR
    tonReq: TON;
END_VAR

Exec();

ACTION HandleBPTM:
// Send the fake BPTM our assertion request by changing stStateReq.stBeamParams
// We expect to recieve bTransitionAuthorized TRUE after some delta T
// We expect bTransitionAuthorized to go FALSE after stMotionStage.bBusy goes FALSE
tonReq(
    IN:=bInTransition,
    PT:=T#3s);
bTransitionAuthorized := tonReq.Q AND stMotionStage.bExecute;
END_ACTION

ACTION HandleFFO:
// Skip implementing this for offline testing
// We won't be able to tell if it worked anyway
END_ACTION

END_FUNCTION_BLOCK

// POUs/Motion/PMPS/FB_Standard_PMPSDB
FUNCTION_BLOCK FB_Standard_PMPSDB
VAR_IN_OUT
    io_fbFFHWO: FB_HardwareFFOutput;
END_VAR
VAR_INPUT
    // If TRUE, FB will run. Reads when enable goes TRUE.
    bEnable: BOOL;
    // E.g. lfe-motion
    sPlcName: STRING;
    {attribute 'pytmc' := '
        pv: REFRESH
        io: io
    '}
    // Set to TRUE to cause an extra read.
    bRefresh: BOOL;
    // Directory where the DB is stored.
    sDirectory: STRING := '/Hard Disk/ftp/PMPS/';
END_VAR
VAR_OUTPUT
    {attribute 'pytmc' := '
        pv: LAST_REFRESH
        io: i
    '}
    nLastRefreshTime: DINT;
    bReadPmpsDb: BOOL;
END_VAR
VAR
    bExecute: BOOL;
    rtEnable: R_TRIG;
    rtRefresh: R_TRIG;
    ftBusy: F_TRIG;

    // Time tracking liften from Arbiter PLCs
    fbTime : FB_LocalSystemTime := ( bEnable := TRUE, dwCycle := 1 );
    fbTime_to_UTC: FB_TzSpecificLocalTimeToSystemTime;
    fbGetTimeZone: FB_GetTimeZoneInformation;
END_VAR

IF NOT bEnable THEN
    RETURN;
END_IF

rtEnable(CLK:=bEnable);
rtRefresh(CLK:=bRefresh);
bRefresh := FALSE;

IF rtEnable.Q OR rtRefresh.Q THEN
    // Make sure file reader gets a rising edge
    MOTION_GVL.fbPmpsFileReader(
        io_fbFFHWO:=io_fbFFHWO,
        bExecute:=FALSE,
    );
    bExecute := TRUE;
END_IF

MOTION_GVL.fbPmpsFileReader(
    io_fbFFHWO:=io_fbFFHWO,
    bExecute:=bExecute,
    sSrcPathName:=CONCAT(CONCAT(sDirectory, sPlcName), '.json'),
    sPLCName:=sPLCName,
    PMPS_jsonDoc=>PMPS_GVL.BP_jsonDoc,
);

ftBusy(CLK:=MOTION_GVL.fbPmpsFileReader.bBusy);
IF ftBusy.Q THEN
    bReadPmpsDb := TRUE;
ELSE
    bReadPmpsDb := FALSE;
END_IF


// Lifted from Arbiter PLCs: keep track of the time
fbTime(sNetID:='');
fbGetTimeZone(sNetID:='', bExecute:=TRUE, tTimeout:=T#10S);
fbTime_to_UTC(in:= fbTime.systemTime , tzInfo:=fbGetTimeZone.tzInfo);

// Update the refresh time on successful read
IF ftBusy.Q AND NOT MOTION_GVL.fbPmpsFileReader.bError THEN
   nLastRefreshTime := TO_DINT(TO_DT(SystemTime_TO_DT(fbTime_to_UTC.out)));
END_IF

bExecute R= ftBusy.Q;

END_FUNCTION_BLOCK

// POUs/Motion/States/Examples/FB_PositionStateInOut
FUNCTION_BLOCK FB_PositionStateInOut EXTENDS FB_PositionStateBase
(*
    Example usage of FB_PositionStateBase for a simple IN/OUT axis. See NOTE: comments.
    Also usable as a drop-in for these cases (no need to roll your own in/out)
*)
VAR_INPUT
    // The enum position to move to
    {attribute 'pytmc' := '
        pv: SET
        io: io
    '}
    enumSet: ENUM_EpicsInOut; // NOTE: Please copy this pragma exactly on your enumSet

    // Information about the OUT position
    stOut: DUT_PositionState; // NOTE: Do not pragma these, let it happen in the manager.
    // Information about the IN position
    stIn: DUT_PositionState;
END_VAR
VAR_OUTPUT
    // The enum state readback
    {attribute 'pytmc' := '
        pv: GET
        io: i
    '}
    enumGet: ENUM_EpicsInOut; // NOTE: Please copy this pragma exactly on your enumGet
END_VAR
VAR
    bInOutInit: BOOL;
END_VAR

IF NOT bInOutInit THEN
    bInOutInit := TRUE;
    arrStates[1] := stOut;
    arrStates[2] := stIn;
    stOut.sName := 'OUT';
    stIn.sName := 'IN';
END_IF
setState := enumSet;
Exec();
enumGet := getState;
enumSet := setState;

END_FUNCTION_BLOCK

// POUs/Motion/States/FB_PositionStateBase
FUNCTION_BLOCK FB_PositionStateBase
(*
    Handles EPICS moves between multiple states for a single axis
    Should be subclassed for a specific enumSet and enumGet.
    See body comment  or FB_PositionStateInOut for an implementation example.
*)
VAR_IN_OUT
    // Motor to move
    stMotionStage: DUT_MotionStage;
END_VAR
VAR_INPUT
    // If TRUE, start a move when setState transitions to a nonzero number
    bEnable: BOOL;
    // On rising edge, reset this FB
    {attribute 'pytmc' := '
        pv: RESET
        io: io
        field: ZNAM False
        field: ONAM True
    '}
    bReset: BOOL;
END_VAR
VAR_OUTPUT
    // If TRUE, there is an error
    {attribute 'pytmc' := '
        pv: ERR
        io: i
        field: ZNAM False
        field: ONAM True
    '}
    bError: BOOL;
    // Error ID
    {attribute 'pytmc' := '
        pv: ERRID
        io: i
    '}
    nErrorId: UDINT;
    // The error that caused bError to flip TRUE
    {attribute 'pytmc' := '
        pv: ERRMSG
        io: i
    '}
    sErrorMessage: STRING;
    // If TRUE, we are moving the motor
    {attribute 'pytmc' := '
        pv: BUSY
        io: i
        field: ZNAM False
        field: ONAM True
    '}
    bBusy: BOOL;
    // If TRUE, we are not moving the motor and the last move completed successfully
    {attribute 'pytmc' := '
        pv: DONE
        io: i
        field: ZNAM False
        field: ONAM True
    '}
    bDone: BOOL;
END_VAR
VAR
    // Pre-allocated array of states
    {attribute 'pytmc' := '
        pv:
        io: io
        expand: %.2d
    '}
    arrStates: ARRAY[1..GeneralConstants.MAX_STATES] OF DUT_PositionState;

    // Corresponding arrStates index to move to, or 0 if no move selected
    setState: INT;
    // The current position we are trying to reach, or 0
    goalState: INT;
    // The readback position
    getState: INT;

    bInit: BOOL;
    stUnknown: DUT_PositionState;
    stGoal: DUT_PositionState;
    fbStateMove: FB_PositionStateMove;
    fbStateInternal: ARRAY[1..GeneralConstants.MAX_STATES] OF FB_PositionStateInternal;
    nIndex: INT;
    bNewGoal: BOOL;
    bInnerExec: BOOL;
    bInnerReset: BOOL;
    rtReset: R_TRIG;
    bMoveRequested: BOOL;
END_VAR

(*
    Subclass me, define enums to translate setState and getState, call Exec

    Example:

    <something to fill arrStates>
    setState := enumSet;
    Exec();
    enumGet := getState;
    enumSet := setState;
*)

ACTION Exec:
StateHandler();
END_ACTION

ACTION StateHandler:
// Reset just goes through the first-cycle init again
rtReset(CLK:=bReset);
IF rtReset.Q THEN
    bInit := FALSE;
    bReset := FALSE;
END_IF

// First-cycle init
IF NOT bInit THEN
    bError := FALSE;
    nErrorID := 0;
    sErrorMessage := '';
    bBusy := FALSE;
    bDone := FALSE;
    bNewGoal := FALSE;
    bInnerExec := FALSE;
    bInnerReset := TRUE;
    setState := 0;
    goalState := 0;
END_IF

// All state internal handlers
FOR nIndex := 1 TO GeneralConstants.MAX_STATES DO
    IF arrStates[nIndex].bValid THEN
        fbStateInternal[nIndex](
            stMotionStage:=stMotionStage,
            stPositionState:=arrStates[nIndex]);
    END_IF
END_FOR

// Check where we are by going through all possible states.
// Note this favors the highest-number state that we're at, it's up to you to make your states mutually exclusive.
getState := 0;
FOR nIndex := 1 TO GeneralConstants.MAX_STATES DO
    IF F_AtPositionState(stMotionStage:=stMotionStage, stPositionState:=arrStates[nIndex]) THEN
        getState := nIndex;
    END_IF
END_FOR

// Use the changing set pv as a rising-edge trigger
IF setState <> goalState THEN
    goalState := setState;
    bNewGoal := TRUE;
END_IF

// Special move handling for error/enable state
IF bError OR NOT bEnable THEN
    bInnerExec := FALSE;
ELSIF bNewGoal THEN
    IF fbStateMove.bBusy THEN
        // Stop previous move if we were already moving but want a new move
        bInnerExec := FALSE;
    ELSE
        // If we hit this branch, we're ready to start a new move
        bInnerExec := TRUE;
        bInnerReset := FALSE;
        bNewGoal := FALSE;
    END_IF
END_IF

// Pick the correct goal structure or Unknown
IF goalState = 0 THEN
    stGoal := stUnknown;
ELSE
    stGoal := arrStates[goalState];
END_IF

// Do the move
fbStateMove(
    stMotionStage := stMotionStage,
    stPositionState := stGoal,
    bExecute := bInnerExec,
    bReset := bInnerReset,
    enumMotionRequest := ENUM_MotionRequest.INTERRUPT,
    bBusy => bBusy);

// Only pass up bDone information if this FB is active
IF bInnerExec THEN
    bDone := fbStateMove.bDone;
END_IF

// Pick up any new errors, but don't override uncleared existing errors
IF NOT bError THEN
    bError := fbStateMove.bError;
    IF bError THEN
        nErrorId := fbStateMove.nErrorId;
        sErrorMessage := fbStateMove.sErrorMessage;
    END_IF
END_IF

// Reset the setpoint and goal to 0 if we're not doing anything
// because FB is waiting for a change from 0 to "something"
bMoveRequested := bInnerExec AND NOT bDone;
IF NOT bError AND NOT bNewGoal AND NOT bMoveRequested THEN
    setState := 0;
    goalState := 0;
    bInnerExec := FALSE;
END_IF

// Bring inner reset back low at the end of the init cycle so that it can be triggered again later
IF NOT bInit THEN
    bInit := TRUE;
    bInnerReset := FALSE;
END_IF
END_ACTION

END_FUNCTION_BLOCK

// POUs/Motion/States/Examples/FB_PositionStateInOut_WithPMPS
FUNCTION_BLOCK FB_PositionStateInOut_WithPMPS EXTENDS FB_PositionStateBase_WithPMPS
(*
    Example usage of FB_PositionStateBase_WithPMPS for a simple IN/OUT axis. See NOTE: comments.
    Also usable as a drop-in for these cases (no need to roll your own in/out)

    This is the PMPS version. Note that the only difference is that we extend the _WithPMPS FB.
*)
VAR_INPUT
    // The enum position to move to
    {attribute 'pytmc' := '
        pv: SET
        io: io
    '}
    enumSet: ENUM_EpicsInOut; // NOTE: Please copy this pragma exactly on your enumSet

    // Information about the OUT position
    stOut: DUT_PositionState; // NOTE: Do not pragma these, let it happen in the manager.
    // Information about the IN position
    stIn: DUT_PositionState;
END_VAR
VAR_OUTPUT
    // The enum state readback
    {attribute 'pytmc' := '
        pv: GET
        io: i
    '}
    enumGet: ENUM_EpicsInOut; // NOTE: Please copy this pragma exactly on your enumGet
END_VAR
VAR
    bInOutInit: BOOL;
END_VAR

IF NOT bInOutInit THEN
    bInOutInit := TRUE;
    arrStates[1] := stOut;
    arrStates[2] := stIn;
    stOut.sName := 'OUT';
    stIn.sName := 'IN';
END_IF
setState := enumSet;
Exec();
enumGet := getState;
enumSet := setState;

END_FUNCTION_BLOCK

// POUs/Motion/States/FB_PositionStateBase_WithPMPS
FUNCTION_BLOCK FB_PositionStateBase_WithPMPS EXTENDS FB_PositionStateBase
(*
    Handles EPICS moves between multiple states for a single axis with PMPS.
    Should be subclassed for a specific enumSet and enumGet.
    See body comment  or FB_PositionStateInOut_WithPMPS for an implementation example.
*)
VAR_IN_OUT
    fbArbiter: FB_Arbiter;
    fbFFHWO: FB_HardwareFFOutput;
END_VAR
VAR_INPUT
    sPmpsDeviceName: STRING;
    sTransitionKey: STRING;
    {attribute 'pytmc' := '
        pv: PMPS:ARB:ENABLE
        io: io
    '}
    bArbiterEnabled: BOOL := TRUE;
    tArbiterTimeout: TIME := T#1s;
    bMoveOnArbiterTimeout: BOOL := TRUE;
    fStateBoundaryDeadband: LREAL := 0;
    bBPOKAutoReset: BOOL := False;
END_VAR
VAR
    {attribute 'pytmc' := 'pv: PMPS'}
    fbStatePMPS: FB_PositionStatePMPS;
    fbEncErrFFO: FB_EncErrorFFO;
END_VAR

(*
    Subclass me, define enums to translate setState and getState, call Exec

    Example:

    <something to fill arrStates>
    setState := enumSet;
    Exec();
    enumGet := getState;
    enumSet := setState;
*)

ACTION Exec:
StateHandler();
PMPSHandler();
END_ACTION

ACTION PMPSHandler:
fbStatePMPS(
    fbArbiter:=fbArbiter,
    fbFFHWO:=fbFFHWO,
    stMotionStage:=stMotionStage,
    arrStates:=arrStates,
    sPmpsDeviceName:=sPmpsDeviceName,
    sTransitionKey:=sTransitionKey,
    stPmpsDoc:= PMPS_GVL.BP_jsonDoc,
    bRequestTransition:=setState <> 0,
    setState:=setState,
    getState:=getState,
    bArbiterEnabled:=bArbiterEnabled,
    tArbiterTimeout:=tArbiterTimeout,
    bMoveOnArbiterTimeout:=bMoveOnArbiterTimeout,
    fStateBoundaryDeadband:=fStateBoundaryDeadband,
    bBPOKAutoReset:=bBPOKAutoReset);

fbEncErrFFO(
    stMotionStage:=stMotionStage,
    fbFFHWO:=fbFFHWO,
    bAutoReset:=TRUE);
END_ACTION

END_FUNCTION_BLOCK

// POUs/Motion/States/Examples/FB_PositionStateInOut_WithPMPS_Test
FUNCTION_BLOCK FB_PositionStateInOut_WithPMPS_Test EXTENDS FB_PositionStateBase_WithPMPS_Test
(*
    Example usage of FB_PositionStateBase_WithPMPS_Test for a simple IN/OUT axis. See NOTE: comments.
    Also usable as a drop-in for these cases (no need to roll your own in/out)

    This is the PMPS version. Note that the only difference is that we extend the _WithPMPS_Test FB.
*)
VAR_INPUT
    // The enum position to move to
    {attribute 'pytmc' := '
        pv: SET
        io: io
    '}
    enumSet: ENUM_EpicsInOut; // NOTE: Please copy this pragma exactly on your enumSet

    // Information about the OUT position
    stOut: DUT_PositionState; // NOTE: Do not pragma these, let it happen in the manager.
    // Information about the IN position
    stIn: DUT_PositionState;
END_VAR
VAR_OUTPUT
    // The enum state readback
    {attribute 'pytmc' := '
        pv: GET
        io: i
    '}
    enumGet: ENUM_EpicsInOut; // NOTE: Please copy this pragma exactly on your enumGet
END_VAR
VAR
    bInOutInit: BOOL;
END_VAR

IF NOT bInOutInit THEN
    bInOutInit := TRUE;
    arrStates[1] := stOut;
    arrStates[2] := stIn;
    stOut.sName := 'OUT';
    stIn.sName := 'IN';
END_IF
setState := enumSet;
Exec();
enumGet := getState;
enumSet := setState;

END_FUNCTION_BLOCK

// POUs/Motion/States/FB_PositionStateBase_WithPMPS_Test
FUNCTION_BLOCK FB_PositionStateBase_WithPMPS_Test EXTENDS FB_PositionStateBase
(*
    Handles EPICS moves between multiple states for a single axis with fake PMPS.
    Should be subclassed for a specific enumSet and enumGet.
    See body comment  or FB_PositionStateInOut_WithPMPS_Test for an implementation example.
*)
VAR_INPUT
    stTransitionBeam: ST_BeamParams := PMPS_GVL.cst0RateBeam;
    nTransitionAssertionID: UDINT;
END_VAR
VAR
    fbStatePMPS: FB_PositionStatePMPS_Test;
END_VAR

(*
    Subclass me, define enums to translate setState and getState, call Exec

    Example:

    <something to fill arrStates>
    setState := enumSet;
    Exec();
    enumGet := getState;
    enumSet := setState;
*)

ACTION Exec:
StateHandler();
PMPSHandler();
END_ACTION

ACTION PMPSHandler:
fbStatePMPS(
    stMotionStage:=stMotionStage,
    arrStates:=arrStates,
    bRequestTransition:=setState <> 0,
    setState:=setState,
    getState:=getState);
END_ACTION

END_FUNCTION_BLOCK

// POUs/Motion/FB_MotionPneumaticActuator
(*This function blcok implements a pnuematic actuator. That can be signle or double acting by setting the ibSingleCntrl accordingly*)
(* with double acting ibCntrlHold signal should be false, while with single acting the signal should be true*)
FUNCTION_BLOCK FB_MotionPneumaticActuator
VAR_INPUT
    (*EPS Interlock Bits*)
    ibInsertOK: BOOL; (*Actuator can be Inserted*)
    ibRetractOK: BOOL; (*ACtuator can be retracted*)
    ibPMPS_OK:BOOL; (*to be linked the Arbiter bit*)
    ibSingleCntrl:BOOL;(* TRUE if Actuator requires one Output signal to be activated, FALSE if its double acting i.e two outputs are required*)
    ibCntrlHold:BOOL; (* Control Signal must retain its value, must be TRUE in the case of single acting*)
    ibOverrideInterlock:BOOL; (*if true interlocks are ignored*)
    // Reset fault
    {attribute 'pytmc' := '
    pv: FFO_Reset
    '}
    i_xReset: BOOL;
    {attribute 'pytmc' := '
    pv: FFO_AutoReset
    '}
    i_xAutoReset: BOOL;
END_VAR
VAR_OUTPUT
    {attribute 'pytmc' := '
    pv:
    '}
    stPneumaticActuator    :    DUT_MotionPneumaticActuator;
    {attribute 'pytmc' := '
     pv: MPS_OK
     field: ZNAM FALSE
     field: ONAM TRUE
     field: DESC TRUE if MPS signal is OK
    '}
    xMPS_OK:BOOL;
END_VAR
VAR_IN_OUT
    io_fbFFHWO    :    FB_HardwareFFOutput;
END_VAR
VAR
    // PMPS
    fbFF    :    FB_FastFault :=(
        i_DevName := 'MPA',
        i_Desc := 'Fault occurs when the device is moving',
        i_TypeCode := 10#1010);

    (*Init*)
    xFirstPass    :    BOOL;
    fbFSInit        :    R_TRIG;

    (* Timeouts*)
    tTimeOutDuration: TIME:= T#10S;
    tInserttimeout: TON;
    tRetracttimeout:TON;
    (*Limit switch latch timer*)
    tLimitSwitchLatchDuration: TIME:=T#1S;
    tInsertLimitSwitch:TON;
    tRetractLimitSwitch:TON;

    (*Logging*)
    fbLogger : FB_LogMessage := (eSubsystem:=E_SubSystem.MOTION);
    ePrevState : ENUM_PnuematicActuatorPositionState;
    tAction : R_TRIG; // Primary action of this device (Insert_DO, Retract_DO, etc.)
    tOverrideActivated : R_TRIG;

    (*IO*)
    i_xInsertedLS    AT%I*: BOOL;
    i_xRetractedLS    AT%I*: BOOL;
    q_xInsert_DO    AT%Q*: BOOL;
    q_xRetract_DO    AT%Q*: BOOL;

END_VAR


(*Initialize*)
fbFSInit( CLK := TRUE, Q => xFirstPass);
IF xFirstPass THEN
    stPneumaticActuator.eState := ENUM_PnuematicActuatorPositionState.INVALID;
    stPneumaticActuator.bRetract_SW := FALSE;
    stPneumaticActuator.bInsert_SW := FALSE;
END_IF

(*Soft IO Mapping to EPICS PVs*)
ACT_IO();

(* Manage States*)
IF stPneumaticActuator.i_bInLimitSwitch AND  stPneumaticActuator.i_bOutLimitSwitch THEN
    stPneumaticActuator.eState:=ENUM_PnuematicActuatorPositionState.INVALID;
ELSIF NOT stPneumaticActuator.i_bInLimitSwitch AND stPneumaticActuator.i_bOutLimitSwitch THEN
    stPneumaticActuator.eState:=ENUM_PnuematicActuatorPositionState.RETRACTED;
ELSIF stPneumaticActuator.i_bInLimitSwitch AND NOT stPneumaticActuator.i_bOutLimitSwitch THEN
    stPneumaticActuator.eState:=ENUM_PnuematicActuatorPositionState.INSERTED;
ELSIF NOT stPneumaticActuator.i_bInLimitSwitch AND NOT stPneumaticActuator.i_bOutLimitSwitch THEN
    stPneumaticActuator.eState:=ENUM_PnuematicActuatorPositionState.MOVING;
ELSE
    stPneumaticActuator.eState:=ENUM_PnuematicActuatorPositionState.INVALID ;
END_IF

(*Set the Done/Busy signal*)
stPneumaticActuator.bDone := (stPneumaticActuator.bRetract_SW AND stPneumaticActuator.eState=ENUM_PnuematicActuatorPositionState.RETRACTED)
                            OR (stPneumaticActuator.bInsert_SW AND stPneumaticActuator.eState=ENUM_PnuematicActuatorPositionState.INSERTED);
stPneumaticActuator.bBusy := (stPneumaticActuator.bRetract_SW AND stPneumaticActuator.eState<>ENUM_PnuematicActuatorPositionState.RETRACTED)
                            OR (stPneumaticActuator.bInsert_SW AND stPneumaticActuator.eState<>ENUM_PnuematicActuatorPositionState.INSERTED);
(*MPS FAULT*)
(* MPS Faults when the actuator is in motion*)
xMPS_OK := (stPneumaticActuator.eState=ENUM_PnuematicActuatorPositionState.RETRACTED) OR (stPneumaticActuator.eState=ENUM_PnuematicActuatorPositionState.INSERTED);
(*PMPS PERMISSION*)
// yet to be implemented

(* Can't have bRetract_SW and  bInsert_SW both be true*)
If (stPneumaticActuator.bRetract_SW) AND (stPneumaticActuator.bInsert_SW) THEN
    stPneumaticActuator.bRetract_SW := FALSE;
    stPneumaticActuator.bInsert_SW := FALSE;
END_IF
//Redundant??
(*Check if both digital outputs active at the same time, and clear all*)
IF stPneumaticActuator.q_bInsert THEN
    stPneumaticActuator.q_bRetract := FALSE;
    stPneumaticActuator.bRetract_SW:= FALSE;
END_IF;
IF stPneumaticActuator.q_bRetract THEN
    stPneumaticActuator.q_bInsert := FALSE;
    stPneumaticActuator.bInsert_SW:= FALSE;
END_IF;

(*Actuate the device*)
stPneumaticActuator.q_bRetract := stPneumaticActuator.bRetractOK AND stPneumaticActuator.bRetract_SW AND NOT stPneumaticActuator.bInsert_SW ;
stPneumaticActuator.q_bInsert := stPneumaticActuator.bInsertOK AND stPneumaticActuator.bInsert_SW AND NOT stPneumaticActuator.bRetract_SW ;

(*Reset the Control signal when command has been executed and give time to ensure the actuator is fully seated in either direction*)
IF (NOT ibSingleCntrl AND NOT ibCntrlHold) THEN
   IF (stPneumaticActuator.bRetract_SW AND stPneumaticActuator.i_bOutLimitSwitch AND tRetractLimitSwitch.Q ) THEN stPneumaticActuator.q_bRetract := FALSE; END_IF
   IF (stPneumaticActuator.bInsert_SW AND stPneumaticActuator.i_bInLimitSwitch AND tInsertLimitSwitch.Q) THEN stPneumaticActuator.q_bInsert := FALSE; END_IF
END_IF

(*Timers*)
tInserttimeout(IN:= stPneumaticActuator.q_bInsert, PT := tTimeOutDuration );
tRetracttimeout(IN:= stPneumaticActuator.q_bRetract, PT := tTimeOutDuration);
tInsertLimitSwitch(IN:= stPneumaticActuator.i_bInLimitSwitch, PT := tLimitSwitchLatchDuration);
tRetractLimitSwitch(IN:= stPneumaticActuator.i_bOutLimitSwitch, PT := tLimitSwitchLatchDuration);


///Check moving postion timout
IF NOT stPneumaticActuator.i_bInLimitSwitch AND tInserttimeout.Q THEN
    stPneumaticActuator.bError := TRUE;
    stPneumaticActuator.sErrorMessage:= 'Actuator insert timeout';
ELSIF NOT stPneumaticActuator.i_bOutLimitSwitch AND tRetracttimeout.Q THEN
    stPneumaticActuator.bError := TRUE;
    stPneumaticActuator.sErrorMessage:= 'Actuator retract timeout';
END_IF
// Reset error
stPneumaticActuator.bError R= stPneumaticActuator.bReset;

(*FAST FAULT*)
fbFF(i_xOK := xMPS_OK,
    i_xReset := i_xReset,
    i_xAutoReset := i_xAutoReset,
    io_fbFFHWO := io_fbFFHWO);

(*Soft IO Mapping to Epics pvs*)
ACT_IO();

ACTION ACT_IO:
(*Inputs*)
stPneumaticActuator.i_bInLimitSwitch :=  i_xInsertedLS;
stPneumaticActuator.i_bOutLimitSwitch := i_xRetractedLS;

(*outputs*)
q_xInsert_DO:=stPneumaticActuator.q_bInsert;
q_xRetract_DO:=stPneumaticActuator.q_bRetract;

(*EPICS*)
stPneumaticActuator.bRetractOK := ibRetractOK;
stPneumaticActuator.bInsertOK := ibInsertOK;
END_ACTION

ACTION ACT_Logger:
// Log Valve timeouts
IF (tInserttimeout.Q OR tRetracttimeout.Q) THEN fbLogger(sMsg:=stPneumaticActuator.sErrorMessage, eSevr:=TcEventSeverity.Warning); END_IF

// Log Actuator commands
// Log valve open
tAction(CLK:= (stPneumaticActuator.q_bRetract OR stPneumaticActuator.q_bInsert));
IF tAction.Q THEN
   IF(stPneumaticActuator.q_bRetract) THEN fbLogger(sMsg:='Actuator commanded retract', eSevr:=TcEventSeverity.Info); END_IF
   IF(stPneumaticActuator.q_bInsert) THEN fbLogger(sMsg:='Actuator commanded insert', eSevr:=TcEventSeverity.Info); END_IF
END_IF


// State Logging
IF ePrevState <> stPneumaticActuator.eState THEN
      CASE stPneumaticActuator.eState OF
        ENUM_PnuematicActuatorPositionState.INVALID:
            fbLogger(sMsg:='Actuator invalid position.', eSevr:=TcEventSeverity.Critical);
          ENUM_PnuematicActuatorPositionState.MOVING:
            fbLogger(sMsg:='Actuator moving', eSevr:=TcEventSeverity.Warning);
        ENUM_PnuematicActuatorPositionState.RETRACTED:
            fbLogger(sMsg:='Actuator Retracted.', eSevr:=TcEventSeverity.Info);
        ENUM_PnuematicActuatorPositionState.INSERTED:
            fbLogger(sMsg:='Actuator Inserted.', eSevr:=TcEventSeverity.Info);
      END_CASE
      ePrevState := stPneumaticActuator.eState;
  END_IF
END_ACTION

END_FUNCTION_BLOCK

// POUs/Motion/FB_MotionStageSim
FUNCTION_BLOCK FB_MotionStageSim
(*
    Set all the values needed for a fake motor to be movable
    via the IOC, then call FB_MotionStage
*)
VAR_IN_OUT
    stMotionStage: DUT_MotionStage;
END_VAR
VAR_INPUT
    nEnableMode: ENUM_StageEnableMode := ENUM_StageEnableMode.ALWAYS;
END_VAR
VAR
    fbMotionStage: FB_MotionStage;
    bInit: BOOL;
END_VAR

IF NOT bInit THEN
    bInit := TRUE;
    // Stand-in for no forward limit
    stMotionStage.bLimitForwardEnable := TRUE;
    // Stand-in for no reverse limit
    stMotionStage.bLimitBackwardEnable := TRUE;
    // Stand-in for no STO button
    stMotionStage.bHardwareEnable := TRUE;
    // Stand-in for no PMPS governer
    stMotionStage.bPowerSelf := TRUE;
    // Always keep it enabled for testing ease
    stMotionStage.nEnableMode := nEnableMode;
END_IF
// Call FB_MotionStage to do the thing
fbMotionStage(stMotionStage := stMotionStage);

END_FUNCTION_BLOCK

// POUs/MotorTesting/FB_MicroStepCountTest
FUNCTION_BLOCK FB_MicroStepCountTest
VAR_INPUT
    bExecute: BOOL;
    fStepSize: LREAL;
    nSteps: UINT;
    fMicroStep: LREAL;
    fVelocity: LREAL;
    tSettleTime: TIME;
END_VAR
VAR_IN_OUT
    Axis: AXIS_REF;
END_VAR
VAR_OUTPUT
    nStepsCounted: UINT;
    nTheorySteps: UINT;
    fPercent: LREAL;
    fEstMicroSize: LREAL;
END_VAR
VAR
    fbMoveRel: MC_MoveRelative;
    fbSettleTimer: TON;
    bDoMove: BOOL;
    nStepCounter: UINT;

    arrPosBuffer: ARRAY [0..99] OF LREAL;
    fAvgPos: LREAL;
    nArrIndex: UINT;
    nLoopIndex: UINT;

    fStartPos: LREAL;
    fPrevPos: LREAL;
    fStepChange: LREAL;

    fStepSum: LREAL;
END_VAR

// Motion FB
fbMoveRel(Axis:=Axis,
    Execute:=bDoMove,
    Distance:=fStepSize,
    Velocity:=fVelocity);

// Settle time
fbSettleTimer(IN:=fbMoveRel.Done,
    PT:=tSettleTime);

// Re-enable the move for next cycle
bDoMove := bExecute AND nStepCounter < nSteps;

// Calculate rolling average
arrPosBuffer[nArrIndex] := Axis.NcToPlc.ActPos;
fAvgPos := 0;
FOR nLoopIndex := 0 TO 99 DO
    fAvgPos := fAvgPos + arrPosBuffer[nLoopIndex];
END_FOR;
fAvgPos := fAvgPos / 100;
nArrIndex := (nArrIndex + 1) MOD 100;

// Initialize starting variables
IF NOT bExecute THEN
    fStartPos := fAvgPos;
    fPrevPos := fAvgPos;
END_IF

// Check results
IF fbSettleTimer.Q THEN
    fStepChange := fAvgPos - fPrevPos;
    // Invert fStepChange if we were doing negative steps
    IF fStepSize < 0 THEN
        fStepChange := fStepChange * -1;
    END_IF
    IF fStepChange > fMicroStep * 0.5 THEN
        nStepsCounted := nStepsCounted + 1;
        fStepSum := fStepSum + fStepChange;
        fEstMicroSize := fStepSum / nStepsCounted;
    END_IF
    nTheorySteps := DINT_TO_UINT(TRUNC(ABS((fStartPos - fAvgPos) / fMicroStep)));
    IF nTheorySteps > 0 THEN
        fPercent := 100 * nStepsCounted / nTheorySteps;
    END_IF
    fPrevPos := fAvgPos;
    nStepCounter := nStepCounter + 1;
    // Reset the move block
    bDoMove := FALSE;
END_IF

END_FUNCTION_BLOCK

// tc_mca_std_lib/POUs/ErrorHandling/FB_ErrorList
FUNCTION_BLOCK FB_ErrorList

VAR_INPUT
	En : BOOL;											//Enable input
	bReset : BOOL;										//Delete all Error entry
	lErrorID : ULINT;									//ErrorID to be acknoledged
	bACK : BOOL;										//Acknoledge the given error and delete it from the list
END_VAR
	
VAR_OUTPUT
	EnO : BOOL;											//Enable output
	nNoError: UINT;										//Number of Errors
	nNoOverflow : INT;									//Number of Overflows
	pErrorSystem : POINTER TO ST_ErrorSystem;			//Pointer to ErrorSystem
END_VAR

VAR
	nFreePos : UINT;									//Number of free position in the list
	nListCnt1 : UINT;									//work variable
	ErrorSystem : ST_ErrorSystem;						//Data structure of the Error list
END_VAR

(*
* ================================================================================
*                                   DESCRIPTION
* ================================================================================
* This Function Block implements the core structure of the Error/Warning Handling
* system. It realizes the datastructure containing every Error Entry, collect
* statistics about the usage and manage the Error Entries.
* Note: The system is under development, most of the functionalities are not
* implemented or existing functionalities may change with time.
* ================================================================================
*)
EnO := En;

//Ponter to ErrorSystem
pErrorSystem := ADR(ErrorSystem);

//Number of overflows
nNoOverflow := ErrorSystem.nNoOverflows;

IF bReset THEN
	MEMSET ( ADR(ErrorSystem.aErrorData[0]), 0, GVL_ErrorSystem.cSizeOfErrorData * SIZEOF(DUT_TerminalError));
	ErrorSystem.lNextErrorID := 1;
END_IF

//Number of errors in the system
nNoError := 0;
FOR nListCnt1 := 0 TO GVL_ErrorSystem.cSizeOfErrorData - 1 DO
	IF ErrorSystem.aErrorData[nListCnt1].Error_ID <> 0  THEN
		nNoError := nNoError+1; 
	END_IF
END_FOR
ErrorSystem.nNoErrors := nNoError;

//Number of free position in the list
nFreePos := GVL_ErrorSystem.cSizeOfErrorData - nNoError;

//Acknoledge specified Error entry
IF bACK THEN
	FOR nListCnt1 := 0 TO GVL_ErrorSystem.cSizeOfErrorData - 1 DO
		IF ErrorSystem.aErrorData[nListCnt1].Error_ID = lErrorID THEN
			ErrorSystem.aErrorData[nListCnt1].ErrorState := DUT_ErrorState.Acknowledged;
		END_IF
	END_FOR
END_IF

//Deleting acknoledged errors
FOR nListCnt1 := 0 TO GVL_ErrorSystem.cSizeOfErrorData - 1 DO
	IF ErrorSystem.aErrorData[nListCnt1].ErrorState = DUT_ErrorState.Acknowledged THEN
		MEMMOVE (ADR(ErrorSystem.aErrorData[nListCnt1]), ADR(ErrorSystem.aErrorData[nListCnt1+1]), (GVL_ErrorSystem.cSizeOfErrorData - 1 - nListCnt1) * SIZEOF(DUT_TerminalError));
		MEMSET(ADR(ErrorSystem.aErrorData[GVL_ErrorSystem.cSizeOfErrorData - 1]), 0, SIZEOF(DUT_TerminalError));
	END_IF
END_FOR

END_FUNCTION_BLOCK

// tc_mca_std_lib/POUs/ErrorHandling/FB_TerminalError
FUNCTION_BLOCK FB_TerminalError

VAR_INPUT
	En					: BOOL;
	iTerminal_ID		: INT;
	bWcState			: BOOL;
	uiInfoData_State	: UINT;
	pErrorSystem		: POINTER TO ST_ErrorSystem;					//Pointer to the error system
END_VAR

VAR_OUTPUT
	EnO : BOOL;
	bError : BOOL := FALSE;
END_VAR

VAR
	iStateError : UINT;
	iOtherError : UINT;
	ErrorData	: DUT_TerminalError;
	nErrSysCNT	: UINT;
	
	//testing
	bStateChanged : BOOL;						//Indicate if state change happened
	uiInfoData_State_Prev : UINT := 16#8;		//Previous value of Infodata.State
	bWcState_Prev : BOOL := FALSE;				//Previous state of WcState
	
	//FB-s
	
END_VAR

(*
Currently:

Problem:

TODO:

*)

//Connect EN to EnO
EnO:=En;

//Check if pointer is OK
IF pErrorSystem=0 THEN RETURN; END_IF

//Any difference from normal state creates an error
IF En AND (bWcState OR uiInfoData_State<>16#8) THEN
	bError:=TRUE;
ELSE
	bError:=FALSE;
END_IF

//Change detection
IF uiInfoData_State <> uiInfoData_State_Prev OR bWcState <> bWcState_Prev THEN
	bStateChanged := TRUE;
ELSE
	bStateChanged := FALSE;
END_IF

//Update previous values
uiInfoData_State_Prev := uiInfoData_State;
bWcState_Prev := bWcState;

//Decision tree
IF bStateChanged THEN
	IF bError THEN
		IF ErrorData.ErrorState = DUT_ErrorState.Active THEN
			//Close active error
			//Read system time
			ErrorData.nDateTimeOff := Tc2_EtherCAT.F_GetActualDcTime64();
			ErrorData.sDateTimeOff := Tc2_EtherCat.DCTIME64_TO_STRING(ErrorData.nDateTimeOff);
			ErrorData.ErrorState := DUT_ErrorState.Inactive;
			//Write Off-time to Error System
			FOR nErrSysCNT := 0 TO GVL_ErrorSystem.cSizeOfErrorData - 1 DO
				IF pErrorSystem^.aErrorData[nErrSysCNT].Error_ID = ErrorData.Error_ID THEN
					pErrorSystem^.aErrorData[nErrSysCNT].nDateTimeOff := ErrorData.nDateTimeOff;
					pErrorSystem^.aErrorData[nErrSysCNT].sDateTimeOff := ErrorData.sDateTimeOff;
					pErrorSystem^.aErrorData[nErrSysCNT].ErrorState := DUT_ErrorState.Inactive;
					EXIT;
				END_IF
			END_FOR
				
			//Clear ErrorData
			MEMSET(ADR(ErrorData), 0, SIZEOF(ErrorData));
		END_IF
		
		//Open a new error
		ErrorData.ErrorState := DUT_ErrorState.Active;												//Set Error State
		ErrorData.nDateTimeOn := Tc2_EtherCAT.F_GetActualDcTime64();								//Get system time
		ErrorData.sDateTimeOn := Tc2_EtherCat.DCTIME64_TO_STRING(ErrorData.nDateTimeOn);			//Convert to string
		ErrorData.iTerminalID := iTerminal_ID;														//Terminal_ID
		ErrorData.bWcState := bWcState;																//WcState bit
		ErrorData.uiInfoDataState := uiInfoData_State;												//uiInfoData_State
		
		//Error message according to uiInfoData_State and WcState
		iStateError := (uiInfoData_State AND 16#000F);												//Mask for operation state 
		iOtherError := (uiInfoData_State AND 16#00F0);												//Mask for the other 3 kind of errors
		//Error messages according to the least significant digit
		CASE iStateError OF
			16#0001 : ErrorData.sErrorMessage := 'Slave in INIT state;   ';
			16#0002 : ErrorData.sErrorMessage := 'Slave in PREOP state;   ';
			16#0003 : ErrorData.sErrorMessage := 'Slave in BOOT state;   ';
			16#0004 : ErrorData.sErrorMessage := 'Slave in SAFEOP state;   ';
			16#0008 : ;																			//Normal operation state
		ELSE
			ErrorData.sErrorMessage := 'Undefined State of operation;   ';						//I hope we will never see this message
			ErrorData.sErrorMessage := CONCAT (ErrorData.sErrorMessage, UINT_TO_STRING(iStateError));
			ErrorData.sErrorMessage := CONCAT (ErrorData.sErrorMessage, '   ');
		END_CASE
		
		//Error messages according to the second least significant digit
		CASE iOtherError OF
			16#0000 : ;																			//No error case
			16#0010 : ErrorData.sErrorMessage := CONCAT (ErrorData.sErrorMessage, 'Slave signals error;   ');
			16#0020 : ErrorData.sErrorMessage := CONCAT (ErrorData.sErrorMessage, 'Invalid vendorID/productCode read;   ');
			16#0040 : ErrorData.sErrorMessage := CONCAT (ErrorData.sErrorMessage, 'Initialisation error occured;   ');
		ELSE
			ErrorData.sErrorMessage := CONCAT (ErrorData.sErrorMessage, 'Undefined Error ID: ');
			ErrorData.sErrorMessage := CONCAT (ErrorData.sErrorMessage, UINT_TO_STRING(iOtherError));
			ErrorData.sErrorMessage := CONCAT (ErrorData.sErrorMessage, '   ');
		END_CASE
	
		//Errormessage according to WcState bit
		IF bWcState THEN
			ErrorData.sErrorMessage := CONCAT (ErrorData.sErrorMessage, 'Invalid Data;');
		END_IF
		
		//Check for overflow
		IF pErrorSystem^.nNoErrors = GVL_ErrorSystem.cSizeOfErrorData THEN
			pErrorSystem^.nNoOverflows := pErrorSystem^.nNoOverflows+1;
		END_IF
		
		//Write Error Data into Error System
		ErrorData.Error_ID := pErrorSystem^.lNextErrorID ;
		MEMMOVE( ADR(pErrorSystem^.aErrorData[1]), ADR(pErrorSystem^.aErrorData[0]), (GVL_ErrorSystem.cSizeOfErrorData-1) * SIZEOF(DUT_TerminalError));
		pErrorSystem^.aErrorData[0] := ErrorData;
		pErrorSystem^.lNextErrorID := pErrorSystem^.lNextErrorID+1;
		
	ELSE
		//Close Active Error
		//Read system time
		ErrorData.nDateTimeOff := Tc2_EtherCAT.F_GetActualDcTime64();
		ErrorData.sDateTimeOff := Tc2_EtherCat.DCTIME64_TO_STRING(ErrorData.nDateTimeOff);
		ErrorData.ErrorState := DUT_ErrorState.Inactive;
		
		//Write Off time to Error System
		FOR nErrSysCNT := 0 TO GVL_ErrorSystem.cSizeOfErrorData - 1 DO
			IF pErrorSystem^.aErrorData[nErrSysCNT].Error_ID = ErrorData.Error_ID THEN
				pErrorSystem^.aErrorData[nErrSysCNT].nDateTimeOff := ErrorData.nDateTimeOff;
				pErrorSystem^.aErrorData[nErrSysCNT].sDateTimeOff := ErrorData.sDateTimeOff;
				pErrorSystem^.aErrorData[nErrSysCNT].ErrorState := DUT_ErrorState.Inactive;
				EXIT;
			END_IF
		END_FOR
			
		//Clear ErrorData
		MEMSET(ADR(ErrorData), 0, SIZEOF(ErrorData));
	END_IF
END_IF

END_FUNCTION_BLOCK

// tc_mca_std_lib/POUs/Hardware/EtherCAT_Terminals/Analog_Inputs/EL3174_0002
//EL3174-0002 | 4-channel analog input, -10/0...+10V, -20/0/+4...20mA, 16 bit, differential
FUNCTION_BLOCK EL3174_0002

VAR_INPUT
	En: BOOL;
	iTerminal_ID : INT;
	ErrorSystem : POINTER TO ST_ErrorSystem;
END_VAR
	
VAR_OUTPUT
	EnO: BOOL;
	iAi_Ch1_Value : INT;
	iAi_Ch2_Value : INT;
	iAi_Ch3_Value : INT;
	iAi_Ch4_Value : INT;
	bError: BOOL;
END_VAR

VAR
	//Channels
	AI_Std_Ch_1_Status	AT %I* : WORD;
	AI_Std_Ch_1_Value 	AT %I* : INT;
	AI_Std_Ch_2_Status 	AT %I* : WORD;
	AI_Std_Ch_2_Value 	AT %I* : INT;
	AI_Std_Ch_3_Status 	AT %I* : WORD;
	AI_Std_Ch_3_Value 	AT %I* : INT;
	AI_Std_Ch_4_Status 	AT %I* : WORD;
	AI_Std_Ch_4_Value 	AT %I* : INT;
	
	//Terminal status
	WcState_WcState AT %I*: BOOL;
	InfoData_State AT %I*: UINT;
	
	//FB-s
	EL3174_0002_Error : FB_TerminalError;
END_VAR

(*
* TODO:
* Status words of the channels
*)

EnO := En;

//Error FB instance
EL3174_0002_Error(
	En := TRUE,
	iTerminal_ID := iTerminal_ID,
	bWcState := WcState_WcState,
	uiInfoData_State := InfoData_State,
	pErrorSystem := ErrorSystem,
	bError => bError,
);

IF En THEN
	IF bError = FALSE THEN
		iAi_Ch1_Value := AI_Std_Ch_1_Value;
		iAi_Ch2_Value := AI_Std_Ch_2_Value;
		iAi_Ch3_Value := AI_Std_Ch_3_Value;
		iAi_Ch4_Value := AI_Std_Ch_4_Value;
	ELSE
		iAi_Ch1_Value := 0;
		iAi_Ch2_Value := 0;
		iAi_Ch3_Value := 0;
		iAi_Ch4_Value := 0;
	END_IF
END_IF

END_FUNCTION_BLOCK

// tc_mca_std_lib/POUs/Hardware/EtherCAT_Terminals/Analog_Inputs/EL3214
//EL3214 | 4-channel analog input terminal, PT100 (RTD)
FUNCTION_BLOCK EL3214

VAR_INPUT
	En: BOOL;
	iTerminal_ID : INT;
	ErrorSystem : POINTER TO ST_ErrorSystem;
END_VAR

VAR_OUTPUT
	EnO: BOOL;
	iAi_Ch1_Value : INT;
	iAi_Ch2_Value : INT;
	iAi_Ch3_Value : INT;
	iAi_Ch4_Value : INT;
	bError: BOOL;
END_VAR

VAR
	//Channels
	AI_RTD_Ch_1_Status	AT %I* : WORD;
	AI_RTD_Ch_1_Value 	AT %I* : INT;
	AI_RTD_Ch_2_Status 	AT %I* : WORD;
	AI_RTD_Ch_2_Value 	AT %I* : INT;
	AI_RTD_Ch_3_Status 	AT %I* : WORD;
	AI_RTD_Ch_3_Value 	AT %I* : INT;
	AI_RTD_Ch_4_Status 	AT %I* : WORD;
	AI_RTD_Ch_4_Value 	AT %I* : INT;
	
	//Terminal status
	WcState_WcState AT %I*: BOOL;
	InfoData_State AT %I*: UINT;
	
	//FB-s
	EL3214_Error : FB_TerminalError;
END_VAR

(*
* TODO:
* Status words of the channels
*)

EnO := En;

//Error FB instance
EL3214_Error(
	En := TRUE,
	iTerminal_ID := iTerminal_ID,
	bWcState := WcState_WcState,
	uiInfoData_State := InfoData_State,
	pErrorSystem := ErrorSystem,
	bError => bError,
);

IF En THEN
	IF bError = FALSE THEN
		iAi_Ch1_Value := AI_RTD_Ch_1_Value;
		iAi_Ch2_Value := AI_RTD_Ch_2_Value;
		iAi_Ch3_Value := AI_RTD_Ch_3_Value;
		iAi_Ch4_Value := AI_RTD_Ch_4_Value;
	ELSE
		iAi_Ch1_Value := 0;
		iAi_Ch2_Value := 0;
		iAi_Ch3_Value := 0;
		iAi_Ch4_Value := 0;
	END_IF
END_IF

END_FUNCTION_BLOCK

// tc_mca_std_lib/POUs/Hardware/EtherCAT_Terminals/Analog_Inputs/EL3255
//EL3255 | 5-channel potentiometer measurement with sensor supply
FUNCTION_BLOCK EL3255

VAR_INPUT
	En: BOOL;
	iTerminal_ID : INT;
	ErrorSystem : POINTER TO ST_ErrorSystem;
END_VAR

VAR_OUTPUT
	EnO : BOOL;	
	Ch1_Value : INT;
	Ch2_Value : INT;
	Ch3_Value : INT;
	Ch4_Value : INT;
	Ch5_Value : INT;
	bError : BOOL;
END_VAR

VAR
	AI_Std_Ch1_Value AT %I* : INT;
	AI_Std_Ch2_Value AT %I* : INT;
	AI_Std_Ch3_Value AT %I* : INT;
	AI_Std_Ch4_Value AT %I* : INT;
	AI_Std_Ch5_Value AT %I* : INT;
	WcState_WcState AT %I*: BOOL;
	InfoData_State AT %I*: UINT;
	
	//FB-s
	EL3255_Error : FB_TerminalError;
END_VAR

(*
* TODO:
* Channel Status words
*)

EnO:=En;

//Error FB instance
EL3255_Error(
	En := TRUE,
	iTerminal_ID := iTerminal_ID,
	bWcState := WcState_WcState,
	uiInfoData_State := InfoData_State,
	pErrorSystem := ErrorSystem,
	bError => bError,
);

IF EN THEN
	IF NOT bError THEN
		Ch1_Value := AI_Std_Ch1_Value;
		Ch2_Value := AI_Std_Ch2_Value;
		Ch3_Value := AI_Std_Ch3_Value;
		Ch4_Value := AI_Std_Ch4_Value;
		Ch5_Value := AI_Std_Ch5_Value;
	ELSE
		Ch1_Value := 0;
		Ch2_Value := 0;
		Ch3_Value := 0;
		Ch4_Value := 0;
		Ch5_Value := 0;
	END_IF
END_IF

END_FUNCTION_BLOCK

// tc_mca_std_lib/POUs/Hardware/EtherCAT_Terminals/Analog_Inputs/FB_CalculateFrequency_3702_v0_01
FUNCTION_BLOCK FB_CalculateFrequency_3702_v0_01
VAR CONSTANT
	///200 samples/period
	cBufferSize: INT := 1000;
END_VAR
VAR_INPUT
	En: BOOL;
	bCalculate: BOOL;
	aBufferValue: ARRAY[0..(cBuffersize - 1)] OF INT;
	aBufferDcTime: ARRAY[0..(cBuffersize - 1)] OF UDINT;
	///If curve has a DC offset
	nDCOffset: INT := 0;
END_VAR
VAR_OUTPUT
	EnO: BOOL;
	bError: BOOL;
	fActFrequency: LREAL;
END_VAR
VAR
	nIndex: INT;
	nFirstZeroCrossing: INT;
	nLastZeroCrossing: INT;
	rTimeFirst: REAL := 0;
	rTimeLast: REAL := 0;
	rTimeRes: REAL := 0;
	nCrossings: INT := 0;
END_VAR
VAR_TEMP
	rRange: REAL := 0;
	rTimeSpan: REAL := 0;
END_VAR

EnO:=En;
bError:=FALSE;
nCrossings:=0;
IF En AND bCalculate THEN
	//Serach for crossings of nDCOffset
	FOR nIndex:=1 TO cBuffersize-1 DO
		IF((aBufferValue[nIndex]>nDCOffset AND aBufferValue[nIndex-1]<=nDCOffset) OR (aBufferValue[nIndex]<nDCOffset AND aBufferValue[nIndex-1]>=nDCOffset))	THEN
			IF(nCrossings=0) THEN
				nFirstZeroCrossing:=nIndex;
			END_IF
			nLastZeroCrossing:=nIndex;
			nCrossings:=nCrossings+1;
		END_IF
	END_FOR	
	
	IF nFirstZeroCrossing < nLastZeroCrossing  AND  nCrossings>2 THEN
		//interpolate zero crossings for higher accuracy
		rTimeRes:=UDINT_TO_REAL(aBufferDcTime[1]-aBufferDcTime[0]); //Buffer must contain more than 2 values
		rRange:=INT_TO_REAL(ABS(aBufferValue[nFirstZeroCrossing-1]-aBufferValue[nFirstZeroCrossing]));
		rTimeFirst:=UDINT_TO_REAL( aBufferDcTime[nFirstZeroCrossing-1])+ABS(INT_TO_REAL(aBufferValue[nFirstZeroCrossing-1])/rRange*rTimeRes);
		rRange:=INT_TO_REAL(ABS(aBufferValue[nLastZeroCrossing-1]-aBufferValue[nLastZeroCrossing]));
		rTimeLast:=UDINT_TO_REAL( aBufferDcTime[nLastZeroCrossing-1])+ABS(INT_TO_REAL(aBufferValue[nLastZeroCrossing-1])/rRange*rTimeRes);

		//Time span first to last (considering that max one time counter overflow have occured in the total time range of the time buffer)	
		IF rTimeFirst<rTimeLast THEN		
			rTimeSpan:=rTimeLast-rTimeFirst;
		ELSE //overflow of counter once (only 32bit timestamp =4.29seconds)
			rTimeSpan:=4294967296.0-rTimeFirst+rTimeLast;
		END_IF
		
		fActFrequency:=1000000000.0/rTimeSpan*(nCrossings-1)/2; //two crossings per period => Average frequency over buffer.
	ELSE
		fActFrequency:=0;
	END_IF
END_IF

END_FUNCTION_BLOCK

// tc_mca_std_lib/POUs/Hardware/EtherCAT_Terminals/Digital_Inputs/EL1008
///EL1008 | 8-channel digital input terminal 24 V DC, 3 ms
FUNCTION_BLOCK EL1008

VAR_INPUT
	En: BOOL;
	iTerminal_ID : INT;
	ErrorSystem : POINTER TO ST_ErrorSystem;
END_VAR

VAR_OUTPUT
	EnO: BOOL;
	bDi_1: BOOL;
	bDi_2: BOOL;
	bDi_3: BOOL;
	bDi_4: BOOL;
	bDi_5: BOOL;
	bDi_6: BOOL;
	bDi_7: BOOL;
	bDi_8: BOOL;
	bError: BOOL;
END_VAR

VAR
	Channel_1_Input AT %I*: BOOL;
	Channel_2_Input AT %I*: BOOL;
	Channel_3_Input AT %I*: BOOL;
	Channel_4_Input AT %I*: BOOL;
	Channel_5_Input AT %I*: BOOL;
	Channel_6_Input AT %I*: BOOL;
	Channel_7_Input AT %I*: BOOL;
	Channel_8_Input AT %I*: BOOL;
	WcState_WcState AT %I*: BOOL;
	InfoData_State AT %I*: UINT;
	
	//FB-s
	EL1008_Error : FB_TerminalError;
END_VAR

EnO:=En;

//Error FB instance
EL1008_Error(
	En := TRUE,
	iTerminal_ID := iTerminal_ID,
	bWcState := WcState_WcState,
	uiInfoData_State := InfoData_State,
	pErrorSystem := ErrorSystem,
	bError => bError,
);

IF En THEN
	IF bError=FALSE THEN
		bDi_1:=Channel_1_Input;
		bDi_2:=Channel_2_Input;
		bDi_3:=Channel_3_Input;
		bDi_4:=Channel_4_Input;
		bDi_5:=Channel_5_Input;
		bDi_6:=Channel_6_Input;
		bDi_7:=Channel_7_Input;
		bDi_8:=Channel_8_Input;
	ELSE
		bDi_1:=FALSE;
		bDi_2:=FALSE;
		bDi_3:=FALSE;
		bDi_4:=FALSE;
		bDi_5:=FALSE;
		bDi_6:=FALSE;
		bDi_7:=FALSE;
		bDi_8:=FALSE;
	END_IF
END_IF

END_FUNCTION_BLOCK

// tc_mca_std_lib/POUs/Hardware/EtherCAT_Terminals/Digital_Inputs/EL1018
///EL1018 | 8-channel digital input terminal 24 V DC, 10 µs
FUNCTION_BLOCK EL1018

VAR_INPUT
	En: BOOL;
	iTerminal_ID : INT;
	ErrorSystem : POINTER TO ST_ErrorSystem;
END_VAR

VAR_OUTPUT
	EnO: BOOL;
	bDi_1: BOOL;
	bDi_2: BOOL;
	bDi_3: BOOL;
	bDi_4: BOOL;
	bDi_5: BOOL;
	bDi_6: BOOL;
	bDi_7: BOOL;
	bDi_8: BOOL;
	bError : BOOL;
END_VAR

VAR
	Channel_1_Input AT %I*: BOOL;
	Channel_2_Input AT %I*: BOOL;
	Channel_3_Input AT %I*: BOOL;
	Channel_4_Input AT %I*: BOOL;
	Channel_5_Input AT %I*: BOOL;
	Channel_6_Input AT %I*: BOOL;
	Channel_7_Input AT %I*: BOOL;
	Channel_8_Input AT %I*: BOOL;
	WcState_WcState AT %I*: BOOL;
	InfoData_State  AT %I*: UINT;
	
	//FB-s
	EL1018_Error : FB_TerminalError;
END_VAR

EnO:=En;

//Error FB instance
EL1018_Error(
	En := TRUE,
	iTerminal_ID := iTerminal_ID,
	bWcState := WcState_WcState,
	uiInfoData_State := InfoData_State,
	pErrorSystem := ErrorSystem,
	bError => bError,
);

IF En THEN
	IF bError=FALSE THEN
		bDi_1:=Channel_1_Input;
		bDi_2:=Channel_2_Input;
		bDi_3:=Channel_3_Input;
		bDi_4:=Channel_4_Input;
		bDi_5:=Channel_5_Input;
		bDi_6:=Channel_6_Input;
		bDi_7:=Channel_7_Input;
		bDi_8:=Channel_8_Input;
	ELSE
		bDi_1:=FALSE;
		bDi_2:=FALSE;
		bDi_3:=FALSE;
		bDi_4:=FALSE;
		bDi_5:=FALSE;
		bDi_6:=FALSE;
		bDi_7:=FALSE;
		bDi_8:=FALSE;
	END_IF
END_IF

END_FUNCTION_BLOCK

// tc_mca_std_lib/POUs/Hardware/EtherCAT_Terminals/Digital_Inputs/EL1808
///EL1808 | HD EtherCAT Terminals, 8-channel digital input 24 V DC, 3 ms, 2-wire connection
FUNCTION_BLOCK EL1808

VAR_INPUT
	En: BOOL;
	iTerminal_ID : INT;
	ErrorSystem : POINTER TO ST_ErrorSystem;
END_VAR

VAR_OUTPUT
	EnO: BOOL;
	bDi_1: BOOL;
	bDi_2: BOOL;
	bDi_3: BOOL;
	bDi_4: BOOL;
	bDi_5: BOOL;
	bDi_6: BOOL;
	bDi_7: BOOL;
	bDi_8: BOOL;
	bError: BOOL;
END_VAR

VAR
	Channel_1_Input AT %I*: BOOL;
	Channel_2_Input AT %I*: BOOL;
	Channel_3_Input AT %I*: BOOL;
	Channel_4_Input AT %I*: BOOL;
	Channel_5_Input AT %I*: BOOL;
	Channel_6_Input AT %I*: BOOL;
	Channel_7_Input AT %I*: BOOL;
	Channel_8_Input AT %I*: BOOL;
	WcState_WcState AT %I*: BOOL;
	InfoData_State AT %I*: UINT;
	
	//FB-s
	EL1808_Error : FB_TerminalError;
END_VAR

EnO:=En;

//Error FB instance
EL1808_Error(
	En := TRUE,
	iTerminal_ID := iTerminal_ID,
	bWcState := WcState_WcState,
	uiInfoData_State := InfoData_State,
	pErrorSystem := ErrorSystem,
	bError => bError,
);

IF En THEN
	IF bError=FALSE THEN
		bDi_1:=Channel_1_Input;
		bDi_2:=Channel_2_Input;
		bDi_3:=Channel_3_Input;
		bDi_4:=Channel_4_Input;
		bDi_5:=Channel_5_Input;
		bDi_6:=Channel_6_Input;
		bDi_7:=Channel_7_Input;
		bDi_8:=Channel_8_Input;
	ELSE
		bDi_1:=FALSE;
		bDi_2:=FALSE;
		bDi_3:=FALSE;
		bDi_4:=FALSE;
		bDi_5:=FALSE;
		bDi_6:=FALSE;
		bDi_7:=FALSE;
		bDi_8:=FALSE;
	END_IF
END_IF

END_FUNCTION_BLOCK

// tc_mca_std_lib/POUs/Hardware/EtherCAT_Terminals/Digital_Inputs/EL1809
///EL1809 | HD EtherCAT Terminals, 16-channel digital input 24 V DC, 3 ms
FUNCTION_BLOCK EL1809

VAR_INPUT
	En: BOOL;
	iTerminal_ID : INT;
	ErrorSystem : POINTER TO ST_ErrorSystem;
END_VAR

VAR_OUTPUT
	EnO: BOOL;
	bDi_1: BOOL;
	bDi_2: BOOL;
	bDi_3: BOOL;
	bDi_4: BOOL;
	bDi_5: BOOL;
	bDi_6: BOOL;
	bDi_7: BOOL;
	bDi_8: BOOL;
	bDi_9: BOOL;
	bDi_10: BOOL;
	bDi_11: BOOL;
	bDi_12: BOOL;
	bDi_13: BOOL;
	bDi_14: BOOL;
	bDi_15: BOOL;
	bDi_16: BOOL;
	bError: BOOL;
END_VAR

VAR
	Channel_1_Input AT %I*: BOOL;
	Channel_2_Input AT %I*: BOOL;
	Channel_3_Input AT %I*: BOOL;
	Channel_4_Input AT %I*: BOOL;
	Channel_5_Input AT %I*: BOOL;
	Channel_6_Input AT %I*: BOOL;
	Channel_7_Input AT %I*: BOOL;
	Channel_8_Input AT %I*: BOOL;
	Channel_9_Input AT %I*: BOOL;
	Channel_10_Input AT %I*: BOOL;
	Channel_11_Input AT %I*: BOOL;
	Channel_12_Input AT %I*: BOOL;
	Channel_13_Input AT %I*: BOOL;
	Channel_14_Input AT %I*: BOOL;
	Channel_15_Input AT %I*: BOOL;
	Channel_16_Input AT %I*: BOOL;
	WcState_WcState AT %I*: BOOL;
	InfoData_State AT %I*: UINT;
	
	//FB-s
	EL1809_Error : FB_TerminalError;
END_VAR

EnO:=En;

//Error FB instance
EL1809_Error(
	En := TRUE,
	iTerminal_ID := iTerminal_ID,
	bWcState := WcState_WcState,
	uiInfoData_State := InfoData_State,
	pErrorSystem := ErrorSystem,
	bError => bError,
);

IF En THEN
	IF bError=FALSE THEN
		bDi_1:=Channel_1_Input;
		bDi_2:=Channel_2_Input;
		bDi_3:=Channel_3_Input;
		bDi_4:=Channel_4_Input;
		bDi_5:=Channel_5_Input;
		bDi_6:=Channel_6_Input;
		bDi_7:=Channel_7_Input;
		bDi_8:=Channel_8_Input;
		bDi_9:=Channel_9_Input;
		bDi_10:=Channel_10_Input;
		bDi_11:=Channel_11_Input;
		bDi_12:=Channel_12_Input;
		bDi_13:=Channel_13_Input;
		bDi_14:=Channel_14_Input;
		bDi_15:=Channel_15_Input;
		bDi_16:=Channel_16_Input;
	ELSE
		bDi_1:=FALSE;
		bDi_2:=FALSE;
		bDi_3:=FALSE;
		bDi_4:=FALSE;
		bDi_5:=FALSE;
		bDi_6:=FALSE;
		bDi_7:=FALSE;
		bDi_8:=FALSE;
		bDi_9:=FALSE;
		bDi_10:=FALSE;
		bDi_11:=FALSE;
		bDi_12:=FALSE;
		bDi_13:=FALSE;
		bDi_14:=FALSE;
		bDi_15:=FALSE;
		bDi_16:=FALSE;
	END_IF
END_IF

END_FUNCTION_BLOCK

// tc_mca_std_lib/POUs/Hardware/EtherCAT_Terminals/Digital_Inputs/EL1819
///EL1819 | HD EtherCAT Terminals, 16-channel digital input 24 V DC, 10 µs
FUNCTION_BLOCK EL1819

VAR_INPUT
	En: BOOL;
	iTerminal_ID : INT;
	ErrorSystem : POINTER TO ST_ErrorSystem;
END_VAR

VAR_OUTPUT
	EnO: BOOL;
	bDi_1: BOOL;
	bDi_2: BOOL;
	bDi_3: BOOL;
	bDi_4: BOOL;
	bDi_5: BOOL;
	bDi_6: BOOL;
	bDi_7: BOOL;
	bDi_8: BOOL;
	bDi_9: BOOL;
	bDi_10: BOOL;
	bDi_11: BOOL;
	bDi_12: BOOL;
	bDi_13: BOOL;
	bDi_14: BOOL;
	bDi_15: BOOL;
	bDi_16: BOOL;
	bError: BOOL;
END_VAR

VAR
	Channel_1_Input AT %I*: BOOL;
	Channel_2_Input AT %I*: BOOL;
	Channel_3_Input AT %I*: BOOL;
	Channel_4_Input AT %I*: BOOL;
	Channel_5_Input AT %I*: BOOL;
	Channel_6_Input AT %I*: BOOL;
	Channel_7_Input AT %I*: BOOL;
	Channel_8_Input AT %I*: BOOL;
	Channel_9_Input AT %I*: BOOL;
	Channel_10_Input AT %I*: BOOL;
	Channel_11_Input AT %I*: BOOL;
	Channel_12_Input AT %I*: BOOL;
	Channel_13_Input AT %I*: BOOL;
	Channel_14_Input AT %I*: BOOL;
	Channel_15_Input AT %I*: BOOL;
	Channel_16_Input AT %I*: BOOL;
	WcState_WcState AT %I*: BOOL;
	InfoData_State AT %I*: UINT;
	
	//FB-s
	EL1819_Error : FB_TerminalError;
END_VAR

EnO:=En;

//Error FB instance
EL1819_Error(
	En := TRUE,
	iTerminal_ID := iTerminal_ID,
	bWcState := WcState_WcState,
	uiInfoData_State := InfoData_State,
	pErrorSystem := ErrorSystem,
	bError => bError,
);

IF En THEN
	IF bError=FALSE THEN
		bDi_1:=Channel_1_Input;
		bDi_2:=Channel_2_Input;
		bDi_3:=Channel_3_Input;
		bDi_4:=Channel_4_Input;
		bDi_5:=Channel_5_Input;
		bDi_6:=Channel_6_Input;
		bDi_7:=Channel_7_Input;
		bDi_8:=Channel_8_Input;
		bDi_9:=Channel_9_Input;
		bDi_10:=Channel_10_Input;
		bDi_11:=Channel_11_Input;
		bDi_12:=Channel_12_Input;
		bDi_13:=Channel_13_Input;
		bDi_14:=Channel_14_Input;
		bDi_15:=Channel_15_Input;
		bDi_16:=Channel_16_Input;
	ELSE
		bDi_1:=FALSE;
		bDi_2:=FALSE;
		bDi_3:=FALSE;
		bDi_4:=FALSE;
		bDi_5:=FALSE;
		bDi_6:=FALSE;
		bDi_7:=FALSE;
		bDi_8:=FALSE;
		bDi_9:=FALSE;
		bDi_10:=FALSE;
		bDi_11:=FALSE;
		bDi_12:=FALSE;
		bDi_13:=FALSE;
		bDi_14:=FALSE;
		bDi_15:=FALSE;
		bDi_16:=FALSE;
	END_IF
END_IF

END_FUNCTION_BLOCK

// tc_mca_std_lib/POUs/Hardware/EtherCAT_Terminals/Digital_Inputs/FB_EL1252ASM_v1_00
FUNCTION_BLOCK FB_EL1252ASM_v1_00
VAR_INPUT
	En: BOOL;
END_VAR
VAR_OUTPUT
	EnO: BOOL;
	Di_1: BOOL;
	Di_2: BOOL;
	Di_1_LatchTimePos: ULINT;
	Di_2_LatchTimePos: ULINT;
	Di_1_LatchTimeNeg: ULINT;
	Di_2_LatchTimeNeg: ULINT;
	///Below bits can be used but then they must be enabled in the COE of the card. Nicklas suggested to not use these (since something wss written that you then only were allowed to read the latch time onece (some kkind of auto reset??))	
	///Di_1_LatchNeg:BOOL;
	///	Di_1_LatchPos:BOOL;
	///	Di_2_LatchNeg:BOOL;
	///	Di_2_LatchPos:BOOL;
	Error: BOOL;
END_VAR
VAR
	Channel_1_Input AT %I*: BOOL;
	Channel_2_Input AT %I*: BOOL;
	///Latch_Status1 AT %I*: USINT;
	///	Latch_Status2 AT %I*: USINT;
	Latch_LatchPos1 AT %I*: ULINT;
	Latch_LatchNeg1 AT %I*: ULINT;
	Latch_LatchPos2 AT %I*: ULINT;
	Latch_LatchNeg2 AT %I*: ULINT;
	WcState_WcState AT %I*: BOOL;
	InfoData_State AT %I*: UINT;
END_VAR

EnO:=En;

IF En AND (WcState_WcState OR InfoData_State<>16#8) THEN //InfoData_State==0 => in OP mode
	Error:=TRUE;
ELSE
	Error:=FALSE;
END_IF

IF En THEN
	IF Error=FALSE THEN
		Di_1:=Channel_1_Input;
		Di_2:=Channel_2_Input;
	(*	Di_1_LatchPos:=Latch_Status1.0;
		Di_1_LatchNeg:=Latch_Status1.1;
		Di_2_LatchPos:=Latch_Status2.0;
		Di_2_LatchNeg:=Latch_Status2.1;*)
		Di_1_LatchTimePos:=Latch_LatchPos1;
		Di_2_LatchTimePos:=Latch_LatchPos2;		
		Di_1_LatchTimeNeg:=Latch_LatchNeg1;		
		Di_2_LatchTimeNeg:=Latch_LatchNeg2;
		
	ELSE
		Di_1:=FALSE;
		Di_2:=FALSE;
	END_IF
END_IF

END_FUNCTION_BLOCK

// tc_mca_std_lib/POUs/Hardware/EtherCAT_Terminals/Digital_Outputs/EL2014
FUNCTION_BLOCK EL2014
VAR_INPUT
	En: BOOL;
	iTerminal_ID : INT; 
	bDo_1: BOOL;
	bDo_2: BOOL;
	bDo_3: BOOL;
	bDo_4: BOOL;
	ErrorSystem : POINTER TO ST_ErrorSystem;
END_VAR

VAR_OUTPUT
	EnO : BOOL;
	bError : BOOL;
END_VAR

